// TwinCAT 3 PLC project Tester_QA
// ProgramVersion: 3.1.4024.0
// libraries:
//   AircomLibrary, * (AirCom)
//   VisuElemBase, * (System)
//   Tc2_Standard, * (Beckhoff Automation GmbH)
//   Tc2_SUPS, * (Beckhoff Automation GmbH)
//   Tc2_System, * (Beckhoff Automation GmbH)
//   Tc2_Utilities, * (Beckhoff Automation GmbH)
//   Tc3_Module, * (Beckhoff Automation GmbH)
//   VisuDialogs, * (System)
//   Visu User Mgmt Interfaces,newest,System
//   VisuSymbols,3.5.10.0,System
// project tree:
//   / GlobalTextList.TcGTLO, PlcTask.TcTTO, Visualization Manager.TcVMO (not stored), VISU_TASK.TcTTO
//   GVLs/ GVL_IO.TcGVL, GVL_TesterParams.TcGVL
//   POUs/ MAIN.TcPOU
//   QATester/MainBlock/Chamber/FB/ fbChamber.TcPOU, fbSaveFiles.TcPOU
//   QATester/MainBlock/Chamber/ST/ nCompresorTypes.TcDUT (not stored), nTestType.TcDUT (not stored), stControl.TcDUT, stInOuts.TcDUT, stParamsChamber.TcDUT, stTestParams.TcDUT (not stored)
//   QATester/MainBlock/ fbMainBlock.TcPOU
//   QATester/VISUs/Common/ MeasureCalibration.TcVIS, vSmallChamber.TcVIS, vSmallChamber_WEB.TcVIS, vSmallChamber_v2.TcVIS, vSmallChamber_v2_WEB.TcVIS, vTestPicker.TcVIS
//   QATester/VISUs/Screens/Connected/ vFileSave.TcVIS (not stored), vPlotScreen.TcVIS, vRecipe.TcVIS, vService.TcVIS (not stored)
//   QATester/VISUs/Screens/HMI/ vMainScreen.TcVIS, vStatusScreen.TcVIS, vStatusScreen_v2.TcVIS
//   QATester/VISUs/Screens/WEB/ vMainScreen_WEB.TcVIS, vStatusScreen_v2_WEB.TcVIS, vStatusScreen_WEB.TcVIS
//   QATester/VISUs/TextLists/ txlCompresorTypes.TcTLO, txlTestTypes.TcTLO
//   QATester/VISUs/ vMain.TcVIS, vMain_WEB.TcVIS
// real-time tasks:
//   TASK PlcTask: cycle T#10ms, priority 20, ADS port 350
//   TASK VISU_TASK: cycle T#200000us, priority 30, ADS port 351
//   TASK Task 5: cycle T#10ms, priority 1, ADS port 352
// I/O:
//   DEVICE Device 1 (EtherCAT) (disabled), AmsNetId 5.33.161.102.2.1
//     RIO1 (EK1100) [EK1100 EtherCAT Coupler (2A E-Bus)]
//       DI1 (EL1008) [EL1008 8Ch. Dig. Input 24V, 3ms]
//       DO1 (EL2008) [EL2008 8Ch. Dig. Output 24V, 0.5A]
//       DO2 (EL2008) [EL2008 8Ch. Dig. Output 24V, 0.5A]
//       DO3 (EL2008) [EL2008 8Ch. Dig. Output 24V, 0.5A]
//       AI1 (EL3314) [EL3314 4Ch. Ana. Input Thermocouple (TC)]
//       AI2 (EL3164) [EL3164 4Ch. Ana. Input 0-10V]
//       AI3 (EL3164) [EL3164 4Ch. Ana. Input 0-10V]
//       AI4 (EL3164) [EL3164 4Ch. Ana. Input 0-10V]
// variable links:
//   Tester_QA/Tester_QA Instance <-> Device 1 (EtherCAT)/RIO1 (EK1100)/AI1 (EL3314)
//     PlcTask Inputs/GVL_IO.arstInOuts[{0..3}].iTemperature <-> TC Inputs Channel {1..4}/Value  (4 links)
//   Tester_QA/Tester_QA Instance <-> Device 1 (EtherCAT)/RIO1 (EK1100)/AI2 (EL3164)
//     PlcTask Inputs/GVL_IO.arstInOuts[0].iCurrentRaw <-> AI Standard Channel 1/Value
//     PlcTask Inputs/GVL_IO.arstInOuts[1].iCurrentRaw <-> AI Standard Channel 3/Value
//     PlcTask Inputs/GVL_IO.arstInOuts[2].iCurrentRaw <-> AI Standard Channel 2/Value
//     PlcTask Inputs/GVL_IO.arstInOuts[3].iCurrentRaw <-> AI Standard Channel 4/Value
//   Tester_QA/Tester_QA Instance <-> Device 1 (EtherCAT)/RIO1 (EK1100)/AI3 (EL3164)
//     PlcTask Inputs/GVL_IO.arstInOuts[0].iVoltageRaw <-> AI Standard Channel 1/Value
//     PlcTask Inputs/GVL_IO.arstInOuts[1].iVoltageRaw <-> AI Standard Channel 3/Value
//     PlcTask Inputs/GVL_IO.arstInOuts[2].iVoltageRaw <-> AI Standard Channel 2/Value
//     PlcTask Inputs/GVL_IO.arstInOuts[3].iVoltageRaw <-> AI Standard Channel 4/Value
//   Tester_QA/Tester_QA Instance <-> Device 1 (EtherCAT)/RIO1 (EK1100)/AI4 (EL3164)
//     PlcTask Inputs/GVL_IO.arstInOuts[0].iPressureRaw <-> AI Standard Channel 1/Value
//     PlcTask Inputs/GVL_IO.arstInOuts[1].iPressureRaw <-> AI Standard Channel 3/Value
//     PlcTask Inputs/GVL_IO.arstInOuts[2].iPressureRaw <-> AI Standard Channel 2/Value
//     PlcTask Inputs/GVL_IO.arstInOuts[3].iPressureRaw <-> AI Standard Channel 4/Value
//   Tester_QA/Tester_QA Instance <-> Device 1 (EtherCAT)/RIO1 (EK1100)/DI1 (EL1008)
//     PlcTask Inputs/GVL_IO.arstInOuts[{0..3}].bOverCurrent <-> Channel {1..7 step 2}/Input  (4 links)
//     PlcTask Inputs/GVL_IO.arstInOuts[{0..3}].bSafety <-> Channel 2/Input  (4 links)
//   Tester_QA/Tester_QA Instance <-> Device 1 (EtherCAT)/RIO1 (EK1100)/DO1 (EL2008)
//     PlcTask Outputs/GVL_IO.arstInOuts[{0..3}].bFanON <-> Channel {2..8 step 2}/Output  (4 links)
//     PlcTask Outputs/GVL_IO.arstInOuts[{0..3}].bPowerON <-> Channel {1..7 step 2}/Output  (4 links)
//   Tester_QA/Tester_QA Instance <-> Device 1 (EtherCAT)/RIO1 (EK1100)/DO2 (EL2008)
//     PlcTask Outputs/GVL_IO.arstInOuts[{0..3}].bBottle40l <-> Channel {2..8 step 2}/Output  (4 links)
//     PlcTask Outputs/GVL_IO.arstInOuts[{0..3}].bPressureIn <-> Channel {1..7 step 2}/Output  (4 links)
//   Tester_QA/Tester_QA Instance <-> Device 1 (EtherCAT)/RIO1 (EK1100)/DO3 (EL2008)
//     PlcTask Outputs/GVL_IO.arstInOuts[{0..3}].bEjectPresure <-> Channel {1..7 step 2}/Output  (4 links)
//     PlcTask Outputs/MAIN.fb.bRealease40lTank <-> Channel 2/Output

CONFIGURATION Tester_QA
    RESOURCE PLC ON TwinCAT3
        TASK PlcTask(INTERVAL := T#10ms, PRIORITY := 20);
        TASK VISU_TASK(INTERVAL := T#200000us, PRIORITY := 30);
        PROGRAM MAIN WITH PlcTask : MAIN;
        PROGRAM VisuElems_Visu_Prg WITH VISU_TASK : VisuElems.Visu_Prg;
    END_RESOURCE
END_CONFIGURATION

// ---- QATester/MainBlock/Chamber/ST/stControl.TcDUT
TYPE stControl :
STRUCT
	bStartPerform			 	: BOOL; 		//Wykonanie startu 
	bStartAllow					: BOOL;			//Pozwolenie na start
	bStopPerform				: BOOL;			//Wykonanie stopu
	iSetTest					: nTestType :=nTestType.testEOL;	//Wybrany program
	bChamberBusy				: BOOL;			//Czy komora pracuje
	bTank40Used					: BOOL;			//Czy zbiornik 40l jest używany
	tActualTime					: TIME;			//Czas wymuszenia testu
	bResetChamber				: BOOL;			//Wykonanie resetu po błędzie;
	bChamberResoult				: BOOL;			//Wynik z jakiegokolwiek testu
	sTestResult					: STRING;		//Wynik testu wyświetlany do HMI
END_STRUCT
END_TYPE

// ---- QATester/MainBlock/Chamber/ST/stInOuts.TcDUT
TYPE stInOuts :
STRUCT
	bOverCurrent		AT %I*	: BOOL;			//Przekroczony prąd
	bSafety				AT %I*	: BOOL;			//Obsługa safety
	bPowerON			AT %Q*	: BOOL;			//Załączenie zasilania
	bFanON				AT %Q*	: BOOL;			//Załączenie wentylatora
	bPressureIn			AT %Q*	: BOOL;			//Dobicie ciśnienia do ustalonwej na manometrze wartości
	bBottle40l			AT %Q*	: BOOL;			//Załączenie testu z butlą 40l
	bEjectPresure		AT %Q*	: BOOL;			//Zrzucenie ciśnienia z butli 1l
	bEjectPresure40		AT %Q*	: BOOL;			//Zrzucenie ciśnmienia z butli 40l
	
	iPressureRaw		AT %I* 	: INT;			//Surowa wartość ciśnienia
	iVoltageRaw			AT %I*	: INT;			//Surowa wartość napięcia
	iCurrentRaw			AT %I*	: INT;			//Surowa wartość prądu
	
	rPressure			 		: REAL;			//Wartość ciśnienia
	rVoltage					: REAL;			//Wartość napięcia
	rCurrent					: REAL;			//Wartość prądu
	rTemperature				: REAL;			//Wartość temperatury
	iTemperature		AT %I*	: INT;			//Wartość temperatury
END_STRUCT
END_TYPE

// ---- QATester/MainBlock/Chamber/ST/stParamsChamber.TcDUT
TYPE stParamsChamber :
STRUCT
//Nazwy testów / kompresorów
	sTestName 			: STRING := 'Test';			//Nazwa dla aktuanie wykonywanego testu
	sCompressorName 	: STRING;					//Nazwa dla kompresora
	sErrorDescription	: STRING;					//Opis aktualnego błędu
	sChamberName		: STRING;					//Nazwa komory dla zapisu plików
	sFileDirectory		: STRING;					//Lokalizacja dla zapisu plików
	sFileName			: STRING;					//Nazwa pliku
//Konfigruacja komory
	iCompresorType		: nCompresorTypes := 1;			//Typ kompresora
	iTestNumber			: INT;						//Numer testu
	rMinimalPressure	: REAL;						//Ciśnienie minimalne dla startu komory 
	//stChamberTestParams	:s stTestParams;				//Parametry testu dla komory
	//Parametryzacja zapisu plików
	bSaveToFile			: BOOL;						//Czy zezwolić na zapis do pliku
	iSaveEveryRecords	: INT;						//Wykonaj zapis co ile rekodrów
	iSampleTime0_150	: INT;						//Okres próbkowania do zapisu
	iSampleTime0_1		: INT;						//Okres próbkowania do zapisu
	iSampleTime1_x		: INT;						//Okres próbkowania do zapisu
	sFileCopyLocation	: STRING;					//Gdzie kopoiwać pliki

//Struktury do sterowania skalowaniem wartości fizycznych
	stPressureSens 		: stMeasurementScalingData;	// Parametry skalowania prądu
	stVoltageSens 		: stMeasurementScalingData;	// Parametry skalowania napięcia
	stCurrenteSens 		: stMeasurementScalingData;	// Parametry skalowania prądu
END_STRUCT
END_TYPE

// ---- GVLs/GVL_IO.TcGVL
{attribute 'qualified_only'}
VAR_GLOBAL
	arstInOuts			: ARRAY[0..3] OF stInOuts;
END_VAR

// ---- GVLs/GVL_TesterParams.TcGVL
{attribute 'qualified_only'}
VAR_GLOBAL PERSISTENT
	arTestParams		: ARRAY[0..3] OF stTestParams;
	arstParams			: ARRAY[0..3] OF stParamschamber;
END_VAR
VAR_GLOBAL
	arstControl			: ARRAY[0..3] OF stControl;
	stData				: stAircomTimeStruct;
END_VAR

// ---- POUs/MAIN.TcPOU
PROGRAM MAIN
VAR
	fb : fbMainBlock;
	fbAircomTime : fbDateAndTimeCalc;
	saveDataPresistent : WritePersistentData;
	fbSavePerform	: TON;
	i : INT;
	arTestParams		: ARRAY[0..3] OF stTestParams;
	arstParams			: ARRAY[0..3] OF stParamschamber;
	bSaveData	: BOOL;
	bInit	: BOOL;
END_VAR

IF NOT bInit THEN
	MEMCPY(destAddr:= ADR(arTestParams), srcAddr:=ADR(GVL_TesterParams.arTestParams)  ,n:= SIZEOF(stTestParams)*4);
	MEMCPY(destAddr:= ADR(arstParams), srcAddr:=ADR(GVL_TesterParams.arstParams)  ,n:= SIZEOF(stParamschamber)*4);
	bInit := TRUE;
END_IF
fb(arstControl	:=GVL_TesterParams.arstControl,
	arstParams	:= GVL_TesterParams.arstParams,
	arstInOuts	:= GVL_IO.arstInOuts,
	stChamberTestParams := GVL_TesterParams.arTestParams);
fbAircomTime();

bSaveData	S= (MEMCMP(pBuf1 := ADR(GVL_TesterParams.arTestParams),pBuf2:= ADR(arTestParams), n:= SIZEOF(stTestParams)*4) <> 0) OR (MEMCMP(pBuf1 := ADR(GVL_TesterParams.arstParams),pBuf2:= ADR(arstParams), n:= SIZEOF(stParamschamber)*4) <> 0);
	
fbSavePerform(IN:=bSaveData ,PT:=T#300S);		
IF fbSavePerform.Q THEN
	saveDataPresistent(NETID:='',PORT:=851,START:=TRUE,TMOUT:=T#2S);
	bSaveData R= TRUE;
	MEMCPY(destAddr:= ADR(arTestParams), srcAddr:=ADR(GVL_TesterParams.arTestParams)  ,n:= SIZEOF(stTestParams)*4);
	MEMCPY(destAddr:= ADR(arstParams), srcAddr:=ADR(GVL_TesterParams.arstParams)  ,n:= SIZEOF(stParamschamber)*4);
ELSE
	saveDataPresistent(START:=FALSE);
END_IF

END_PROGRAM

// ---- QATester/MainBlock/fbMainBlock.TcPOU
FUNCTION_BLOCK fbMainBlock
VAR_INPUT
END_VAR
VAR_OUTPUT
END_VAR
VAR_IN_OUT
	arstControl			: ARRAY[0..3] OF stControl;
	arstParams			: ARRAY[0..3] OF stParamschamber;
	arstInOuts			: ARRAY[0..3] OF stInOuts;
	stChamberTestParams : ARRAY[0..3] OF stTestParams;
END_VAR
VAR
	arFbChamber		: ARRAY[0..3] OF fbChamber;
	i			: INT;
	bTankBusy		: BOOL;
	bRealease40lTank	AT %Q* : BOOL;
END_VAR

//Bloki funkcyjne

FOR i := 0 TO 3 DO
	arstControl[i].bStartAllow := NOT arstControl[i].bChamberBusy;		
	arFbChamber[i](stControl:=arstControl[i],stInOuts:=arstInOuts[i],stParams:=arstParams[i],stChamberTestParams:=stChamberTestParams[arstParams[i].iCompresorType],stTime:=GVL_Aircom.stAC_DT_Data);
END_FOR

END_FUNCTION_BLOCK

// ---- QATester/MainBlock/Chamber/FB/fbChamber.TcPOU
FUNCTION_BLOCK fbChamber
VAR_INPUT
END_VAR
VAR_OUTPUT
END_VAR
VAR_IN_OUT
	stControl				: stControl;
	stInOuts 				: stInOuts;
	stParams				: stParamsChamber;
	stChamberTestParams		: stTestParams;
	stTime					: stAircomTimeStruct;	//Struktura czasu
END_VAR
VAR
	//Bloki skalujące
	fbPressureScaller 		:fbAnalogMeasurement;	//Blok skalujący ciśnienie
	fbVoltageScaller	 	:fbAnalogMeasurement;	//Blok skalujący napięcie
	fbCurrentScaller 		:fbAnalogMeasurement;	//Blok skalujący prąd
	iWorkStep : INT;
	//Detekcja prądu
	fbCurrentCheckDelayer	: TON;					//Zwłoka dla wykrywania prądu minimalnego
	//Test EOL
	fbTestTimerEOL			: TON;					//Licznik czasu trwania testu EOL
	bEolTestResult			: BOOL;					//Wynik z testu EOL
	//Test Performance
	fbTestTimerPerformance	: TON;					//Licznik czasu trwania testu Wydajnoiściowego
	bPerfornamceTestResult	: BOOL;					//Wynik z testu Wydajnościowego
	//Test Hour
	fbTestTimerHour	: TON;							//Licznik czasu trwania testu Wydajnoiściowego
	bHourTestResult	: BOOL;							//Wynik z testu Wydajnościowego
	bPressureObtainedHour :BOOL;					//Pierwsza faza zakończona osiągnięto ciśnienie testowe
	//Test Whole
	iWorkStepWhole	: INT;							//Kroki programowe dla testu całościowego
	fbTestTimerWholeI	: TON;							//Licznik czasu I test całkowity
	fbTestTimerWholeII	: TON;							//Licznik czasu II test całkowity
	//Test Under Presure
	bUnderPresureTestResult : BOOL;					//Wynik testu pod ciśnieniem
	rStartUnderPresureLastPresureRecord : REAL;		//Save value of presure before test
	fbUnderPresureTestTimer	: TON;							//Licznik czasu dla tesu pod ciśnieniem
	//Test Cyclic 30
	iCyclicLoopVariable 		: INT;				//Wariable for calculate of cyclic loops
	fbTestTimerCyclic30			: TON;				//Licznik czasu trwania testu cyklicznego 30
	bCyclic30TestResult			: BOOL;				//Wynik testu cyklicznego x30
	fbTestTimerCyclic30On		: TON;				//Timer dla obsługi testu
	bFirstCycle30				: BOOL;				//First cycle indefiner
	iWorkStepTest30				: INT;				//Workstep dla testu cyklicznego 70
	//Test Cyclic 70
	fbTestTimerCyclic70			: TON;				//Licznik czasu trwania testu cyklicznego 30
	bCyclic70TestResult			: BOOL;				//Wynik testu cyklicznego x30
	fbTestTimerCyclic70On		: TON;				//Timer dla obsługi testu
	bFirstCycle70				: BOOL;				//First cycle indefiner
	iWorkStepTest70				: INT;				//Workstep dla testu cyklicznego 70
	//Zmienne do obsługi zapisu plików
	sData						: STRING;			//Data dopisana do lokalizacji
	sDate						: STRING;			//Data rozpoczęcia testu
	sTime						: STRING;			//Godzina rozpoczęcia testu
	sTestName					: STRING;			//Nazwa Test
	sFirstLine					: STRING;			//Dane do zapisu w pierwszej linijce
	sDataString					: STRING(5000);			//dane z pomiarami
	sDataStringTmp				: STRING(5000);			//dane z pomiarami
	sDataStringTmpSave			: STRING(5000);			//Dane do zapisu
	sActualTestTime				: STRING;			//Aktualny czas testu
	sActualPresure				: STRING;			//Aktualna wartość ciśnienia
	sActualVoltage				: STRING;			//Aktualna wartość napięcia
	sActualCurrent				: STRING;			//Aktualna wartość prądu
	sActualTemperature			: STRING;			//Aktualna wartość temperatury
	fbTestTime					: TON;				//Czas wykonywania testu
	iSaveFileRecords			: INT;				//Aktualnie zapisane rekody do zapisu pliku
	iSaveFileRecordsTmp			: INT;				//Zapisana ilość rekordów w tablicy do zapisu (zmienne skopiowane)
	bCreateFile					: BOOL;				//Wymueszenie utworzenia nowego pliku
	bInsertNewStartRows			: BOOL;				//Wymuszenie wstawienia pierwszych 2 wierszy 
	bSavePerform				: BOOL;				//Wykonaj zapis do pliku
	bCopyArray					: BOOL;				//Przygotowanie buforów do zapisu
	arTmpData					: ARRAY[0..1000] OF STRING;	//Tablica z zmiennymi
	arTmpDataCpy				: ARRAY[0..1000] OF STRING;	//Tablica z zmiennymi skopiowanymi
	fbFileOpen					: FB_FileOpen;		//Funkcja dla otwierania pliku
	fbFileClose					: FB_FileClose;		//Funkcja dla zamknięcia pliku
	fbFileWrite					: FB_FileWrite;		//Funkcja dla zapisu pliku
	sFileNameToSave				: STRING;			//Nazwa do zapisu pliku
	bReadyToWrite				: BOOL;				//Zezwolenie na zapis do pliku
	bReadyToClose				: BOOL;				//Zezwolenie na zamknięcie pliku
	bFileSaveError				: BOOL;				//Błąd podczas tworzenie zapisów
	iSampleRecorder				: INT;				//Obsługa samplingu
	fbTestTimer					: TON;				//Obsługa czasu trwania testu
	sTimeRep					: STRING;			//Zmienna dla obsługi czasu godzina 
	fbRiseEdgeError				: R_TRIG;
	iSaveCalc					: INT;				// zmienna pomocnicza podczas zapisu danych
	bRecordTaker				: BOOL;				//Zmienna dla obsługi zbierania danych
	wRecordCalc					: DWORD;			//Zmienna dla lcizenia czasu testu
	bFileCopy					: BOOL;				//Zmienna wykorzystywana podczas kopiowania plików
	fbFileSave					: fbSaveFiles;		//Save files save
	fbFileSaveCopy				: fbSaveFiles;		//Save files save
	//Zmienne dla obsługi rysowania grafów
	arPlotPresure				: ARRAY[0..1000] OF REAL;
	arPlotVoltage				: ARRAY[0..1000] OF REAL;
	arPlotCurrent				: ARRAY[0..1000] OF REAL;
	iPlotRecordCounter			: INT;
	sStepDescription			: STRING;
	iPlotFilter					: INT;
	sFileCopyCommand			: STRING(1000);
	sTemString					: STRING;
	bTEST: BOOL;
	sDirCopy: STRING;
	sPathCopy:STRING;
	iLastWorkStep: INT;
	fbRestON: TON;
END_VAR

ACT_Background();
CASE iWorkStep OF
 0: 				//Inicalizacja
 	iWorkStep := 5;
	stParams.sErrorDescription :='';
	fbTestTimer(IN:=FALSE);
	stInOuts.bFanON := stInOuts.bPowerON := stInOuts.bEjectPresure40 := stInOuts.bEjectPresure := stInOuts.bBottle40l := stInOuts.bPressureIn := FALSE;
 5:					//Idle
 	sStepDescription := 'Chamber Idle';
	stParams.sTestName:= '';
	stControl.tActualTime := T#40D;
	bUnderPresureTestResult R= bCyclic70TestResult R= bCyclic30TestResult R= bPerfornamceTestResult R= bEolTestResult R= stControl.bStartPerform;
 	IF stControl.bStartPerform AND stControl.iSetTest >= 20 AND stInOuts.rPressure <= stParams.rMinimalPressure THEN
		iWorkStep := 6;
		stControl.sTestResult := '';
		stControl.tActualTime := stTime.tActualTime;
	ELSIF stControl.bStartPerform AND stControl.iSetTest = nTestType.testEOL AND stInOuts.rPressure <= stParams.rMinimalPressure THEN
		iWorkStep := stControl.iSetTest;
		stControl.bStartPerform := FALSE;
		bInsertNewStartRows := TRUE;
	ELSIF stControl.bStartPerform THEN
		stInOuts.bEjectPresure := TRUE;
		sStepDescription := 'Presure droping';
	END_IF
 6:
 	sStepDescription := 'Wait for bottle 40l';
 	IF stControl.iSetTest = nTestType.testEOL OR NOT stControl.bStartPerform THEN
		iWorkStep := 5;
		stControl.bStartPerform := FALSE;
		stControl.tActualTime := T#40D;
	END_IF
 	IF stControl.bStartAllow THEN
		bInsertNewStartRows := TRUE;
		bUnderPresureTestResult := bCyclic70TestResult := bCyclic30TestResult := bPerfornamceTestResult := bEolTestResult := FALSE;
		iWorkStep := stControl.iSetTest;
		bFirstCycle70 := bFirstCycle30 := TRUE;
		stControl.bStartAllow := FALSE;
		stControl.bStartPerform := FALSE;
	END_IF

 10: 				//EOL Test
 	stParams.sTestName:= 'EOL_Test';
	ACT_EolTest();
	IF bEolTestResult THEN
		iWorkStep := 1000;
		bEolTestResult:= FALSE;
	END_IF
 20:				//Performance Test
	stParams.sTestName:= 'Performance_Test';
 	ACT_PerformanceTest();
	IF bPerfornamceTestResult THEN
		iWorkStep := 1000;
		bPerfornamceTestResult := FALSE;
	END_IF
 30:				//Hour Test
 	stParams.sTestName:= 'Hour_Test';
 	ACT_HourTest();
	IF bHourTestResult THEN
		iWorkStep := 1000;
		bHourTestResult := FALSE;
	END_IF
 40:				//Whole Test
 	stParams.sTestName:= 'Full_Test';
 	Act_WholeTest();
 50:				//Cyclic x30 Test
 	stParams.sTestName:= 'Cyclic_x30_Test';
 	ACT_Cyclic30Test();
	IF bCyclic30TestResult THEN
		iWorkStep := 1000;
		bCyclic30TestResult := FALSE;
	END_IF
 60:				//Cyclic x70 Test
 	stParams.sTestName:= 'Cyclic_x70_Test';
 	ACT_Cyclic70Test();
	IF bCyclic70TestResult THEN
		iWorkStep := 1000;
		bCyclic70TestResult := FALSE;
	END_IF
 200:				// Błąd
 	//Wysterowanie Timerów i zmiennch
 	fbTestTimerEOL(IN:=FALSE);fbTestTimerPerformance(IN:=FALSE);fbTestTimerHour(IN:=FALSE);fbTestTimerWholeI(IN:=FALSE);
	fbTestTimerWholeII(IN:=FALSE);fbUnderPresureTestTimer(IN:=FALSE);fbTestTimerCyclic30(IN:=FALSE);fbTestTimerCyclic30On(IN:=FALSE);
	fbTestTimerCyclic70(IN:=FALSE);fbTestTimerCyclic70On(IN:=FALSE);
	bUnderPresureTestResult := bCyclic70TestResult := bCyclic30TestResult := bPerfornamceTestResult := bEolTestResult := stInOuts.bFanON := stInOuts.bPowerON := stInOuts.bEjectPresure := stInOuts.bBottle40l := stInOuts.bPressureIn := FALSE;
 	stControl.tActualTime := T#40D;
	stControl.sTestResult := 'Faliure';
 	fbTestTimer(IN:=FALSE);
	stControl.bStartAllow := stControl.bStartPerform := FALSE;
	IF stInOuts.rPressure >= stParams.rMinimalPressure THEN
		stInOuts.bEjectPresure40 := TRUE;
		sStepDescription := 'Error pressure droping';
	ELSE
		stControl.bTank40Used := FALSE;
		stInOuts.bEjectPresure40 := FALSE;
		sStepDescription := 'Wait for reset';
	END_IF
 	IF stControl.bResetChamber THEN
		iWorkStep:=0;
		stControl.bResetChamber := FALSE;
		bFileCopy := TRUE;
	END_IF
 1000:				//Przygotowanie komory do następnego testu
 	stInOuts.bEjectPresure40 S= (bPerfornamceTestResult OR bHourTestResult OR bCyclic70TestResult OR bCyclic30TestResult);
	stInOuts.bEjectPresure S= bEolTestResult;
	iWorkStepTest70 := iWorkStepTest30 := iWorkStepWhole := 0;
	sStepDescription := 'Presure droping';
	stControl.sTestResult := 'DONE';
 	IF stInOuts.rPressure <= stParams.rMinimalPressure THEN
		stControl.tActualTime := T#40D;
		stInOuts.bEjectPresure40 := stInOuts.bEjectPresure := FALSE;
		bUnderPresureTestResult := bCyclic70TestResult := bPerfornamceTestResult := bHourTestResult := bCyclic30TestResult := FALSE;
		iWorkStep := 0;
		bFileCopy := TRUE;
	END_IF
END_CASE

ACTION ACT_Background:
//Obsługa zatrzymania
IF stControl.bChamberBusy AND stControl.bStopPerform THEN
	iWorkStep := 200;
	stControl.bStopPerform := FALSE;
	stParams.sErrorDescription:='Test detained';
END_IF
fbRestON(IN:=stControl.bResetChamber,Pt:=T#200MS);
IF fbRestON.Q THEN
	stControl.bResetChamber  := FALSE;
END_IF
//Skalowanie pomiarów Ciśnienia/Napięcia/Prądu
	fbPressureScaller(rIn:=stInOuts.iPressureRaw,stMeasureScalingData:=stParams.stPressureSens,tStalaCzasowa:=T#10MS,rOutFiltered=>stInOuts.rPressure);
	fbVoltageScaller(rIn:=stInOuts.iVoltageRaw,stMeasureScalingData:=stParams.stVoltageSens,tStalaCzasowa:=T#10MS,rOutFiltered=>stInOuts.rVoltage);
	fbCurrentScaller (rIn:=stInOuts.iCurrentRaw,stMeasureScalingData:=stParams.stCurrenteSens,tStalaCzasowa:=T#10MS,rOutFiltered=>stInOuts.rCurrent);
	stInOuts.rTemperature := stInOuts.iTemperature/10;
//Obsługa Safety
IF stInOuts.bSafety	THEN
	stParams.sErrorDescription := 'Emergency button pressed';
	iWorkStep := 200;
END_IF
//Obsługa daty
sData := CONCAT(WORD_TO_STRING(stTime.stTimeStruct.wYear),'_');
sData := CONCAT(sData,WORD_TO_STRING(stTime.stTimeStruct.wMonth));
//Obsługa zbiornika
	stControl.bTank40Used := iWorkStep >= 20; 		//Określenie czy zbiornik 40l jest wykorzystywany
//Obsługa sekwencji
	stControl.bChamberBusy := (iWorkStep >=10);		//Określenie czy komora wykonuje prace
	stControl.bStartPerform R= (iWorkStep > 6);	//Kasowanie wymuszenia staru po rozpoczęciu nowej pracy
//Sprawowanie kontroli nad prądem minimalnym
	fbCurrentCheckDelayer(IN:=stInOuts.bPowerON,PT:=REAL_TO_TIME(stChamberTestParams.rMinimalCurrentCheckDelay*1000));
	IF fbCurrentCheckDelayer.Q AND (stChamberTestParams.rMinimalCurrentLimit > stInOuts.rCurrent) THEN
		stParams.sErrorDescription := 'Minimal current obtain error';
		iWorkStep := 200;
	END_IF
//Zapis Pliku 
sDate := CONCAT(CONCAT(CONCAT(CONCAT(WORD_TO_STRING(stTime.stTimeStruct.wYear),'_'),WORD_TO_STRING(stTime.stTimeStruct.wMonth)),'_'),WORD_TO_STRING(stTime.stTimeStruct.wDay));
sTimeRep := CONCAT(CONCAT(CONCAT(CONCAT(WORD_TO_STRING(stTime.stTimeStruct.wHour),'_'),WORD_TO_STRING(stTime.stTimeStruct.wMinute)),'_'),WORD_TO_STRING(stTime.stTimeStruct.wSecond));	
sDate := CONCAT(CONCAT(sDate,'_'),sTimeRep);
IF stControl.bChamberBusy AND stParams.bSaveToFile THEN
	ACT_DataSampling();
ELSE
	wRecordCalc := 0;
END_IF
IF stControl.bChamberBusy AND (stParams.sErrorDescription = '') THEN
	ACT_GraphWriter();
	sStepDescription := 'Work in progress';
ELSIF iPlotRecordCounter <> 0 THEN
	iPlotRecordCounter := 0;
	MEMSET(destAddr:=ADR(arPlotPresure),fillByte:=16#00,n:=SIZEOF(arPlotPresure[0])*1000);
	MEMSET(destAddr:=ADR(arPlotVoltage),fillByte:=16#00,n:=SIZEOF(arPlotVoltage[0])*1000);
	MEMSET(destAddr:=ADR(arPlotCurrent),fillByte:=16#00,n:=SIZEOF(arPlotCurrent[0])*1000);
ELSIF NOT stControl.bChamberBusy AND stParams.sErrorDescription = '' THEN
	sStepDescription := 'Idle';
ELSIF stParams.sErrorDescription <> '' THEN
	sStepDescription := 'Chamber Error';
END_IF
//Timer dla obsługi aktualnego czasu
fbTestTime(IN:=stControl.bChamberBusy,PT:=T#5D);
//Wyniki z testów
stControl.bChamberResoult := bUnderPresureTestResult OR bCyclic70TestResult OR bCyclic30TestResult OR bPerfornamceTestResult OR bEolTestResult;
END_ACTION

ACTION ACT_Cyclic30Test:
//Nowa sekwencja
//Obliczanie czasu trwania testu
fbTestTimer(IN:=stINOuts.bPowerON,PT:=T#10D);
//Sekwencja
CASE iWorkStepTest30 OF
	0:	//Test wydajnościowy
		bCyclic30TestResult:= FALSE;
		iCyclicLoopVariable := 0;
		ACT_PerformanceTest();
		IF bPerfornamceTestResult THEN
			iWorkStepTest30 := 10;
		END_IF
	10: //Krok statowy spuszczenie ciśnienia
		bPerfornamceTestResult := FALSE;
		stInOuts.bEjectPresure40 := stInOuts.bEjectPresure := TRUE;
		IF stInOuts.rPressure <= stPArams.rMinimalPressure THEN
			iWorkStepTest30 := 20;
		END_IF
	20:	//Oczekiwanie na dostarczenie do układu ciśnienia po zakończeniu czasu oczekiwania
		stInOuts.bEjectPresure40 := stInOuts.bEjectPresure := FALSE;
		fbTestTimerCyclic30On(IN:=TRUE,PT:=REAL_TO_TIME(stChamberTestParams.rTestCycle30CoolingTime*1000));
		IF fbTestTimerCyclic30On.Q OR bFirstCycle70 THEN
			stInOuts.bPressureIn := TRUE;
		END_IF
		IF stInOuts.bPressureIn AND ABS((stInOuts.rPressure - stChamberTestParams.rStartPresureCycle30Test) < 0.1) THEN
			stInOuts.bPressureIn := FALSE;
			iWorkStepTest70 := 30;
		END_IF
	30:	//Sprawdzenie ciśnienia
		IF stInOuts.bPressureIn AND ((stInOuts.rPressure - stChamberTestParams.rStartPresureCycle30Test) > 0.2) AND stChamberTestParams.bCheckStartPresureCycle70 THEN
			iWorkStep:= 200;
			stInOuts.bFanON := stInOuts.bPowerON := FALSE;
			stInOuts.bEjectPresure40 := stInOuts.bEjectPresure := TRUE;
			stParams.sErrorDescription := 'Wrong start pressure';
			fbTestTimerPerformance(IN:=FALSE);
		ELSE
			iWorkStepTest30 := 40;
		END_IF
	40:	// Rozpoczęcie pierwszej sekwencji
		stInOuts.bFanON := stInOuts.bPowerON := TRUE;
		fbTestTimerCyclic30On(IN:= stInOuts.bPowerON,PT:=REAL_TO_TIME(stChamberTestParams.rTestCycle30LimitTime)*1000);
		IF fbTestTimerCyclic30On.Q AND stChamberTestParams.rPresureToObtainCycle30Test <= stInOuts.rPressure THEN
			iCyclicLoopVariable := iCyclicLoopVariable + 1;
			bFirstCycle30 := FALSE;
			stInOuts.bEjectPresure40 := stInOuts.bEjectPresure := TRUE;
			stInOuts.bPowerON := FALSE;
			fbTestTimerCyclic30On(IN:=FALSE);
			fbTestTimerCyclic30(IN:=FALSE);
			stInOuts.bPowerON := FALSE;
			IF iCyclicLoopVariable >=30 THEN
				iWorkStepTest30 := 50;
				//
				iCyclicLoopVariable := 0;
				bFirstCycle30:= TRUE;
			ELSE
				iWorkStepTest30 := 10;
			END_IF
		END_IF
		IF (fbTestTimerPerformance.Q AND stChamberTestParams.rPresureToObtainCycle70Test >= stInOuts.rPressure) THEN
			iWorkStep:= 200;
			stInOuts.bFanON := stInOuts.bPowerON := FALSE;
			stInOuts.bEjectPresure40 := stInOuts.bEjectPresure := TRUE;
			stParams.sErrorDescription := 'Compressor did not obtain set pressure in limited time';
			bPerfornamceTestResult := FALSE;
			fbTestTimerPerformance(IN:=FALSE);
		END_IF
	50://Zakończenie testu i wykonanie nowego testu wydajnościowego
		bCyclic30TestResult:= FALSE;
		iCyclicLoopVariable := 0;
		ACT_PerformanceTest();
		IF bPerfornamceTestResult THEN
			iWorkStepTest30 := 60;
		END_IF
	60: //Wydanie danych o zakończonej poprawnej pracy
		bCyclic30TestResult := TRUE;
		bPerfornamceTestResult := FALSE;
		fbTestTimerPerformance(IN:=FALSE);
END_CASE
END_ACTION

ACTION ACT_Cyclic70Test:
//Nowa sekwencja
//Obliczanie czasu trwania testu
fbTestTimer(IN:=stINOuts.bPowerON,PT:=T#10D);
//Sekwencja
CASE iWorkStepTest70 OF
	0:	//Test wydajnościowy
		bCyclic70TestResult:= FALSE;
		iCyclicLoopVariable := 0;
		ACT_PerformanceTest();
		IF bPerfornamceTestResult THEN
			iWorkStepTest70 := 10;
		END_IF
	10: //Krok statowy spuszczenie ciśnienia
		bPerfornamceTestResult := FALSE;
		stInOuts.bEjectPresure40 := stInOuts.bEjectPresure := TRUE;
		IF stInOuts.rPressure <= stPArams.rMinimalPressure THEN
			iWorkStepTest70 := 20;
		END_IF
	20:	//Oczekiwanie na dostarczenie do układu ciśnienia po zakończeniu czasu oczekiwania
		stInOuts.bEjectPresure40 := stInOuts.bEjectPresure := FALSE;
		fbTestTimerCyclic70On(IN:=TRUE,PT:=REAL_TO_TIME(stChamberTestParams.rTestCycle70CoolingTime*1000));
		IF fbTestTimerCyclic70On.Q OR bFirstCycle70 THEN
			stInOuts.bPressureIn := TRUE;
		END_IF
		IF stInOuts.bPressureIn AND ABS((stInOuts.rPressure - stChamberTestParams.rStartPresureCycle70Test) < 0.1) THEN
			stInOuts.bPressureIn := FALSE;
			iWorkStepTest70 := 30;
		END_IF
	30:	//Sprawdzenie ciśnienia
		IF stInOuts.bPressureIn AND ((stInOuts.rPressure - stChamberTestParams.rStartPresureCycle70Test) > 0.2) AND stChamberTestParams.bCheckStartPresureCycle70 THEN
			iWorkStep:= 200;
			stInOuts.bFanON := stInOuts.bPowerON := FALSE;
			stInOuts.bEjectPresure40 := stInOuts.bEjectPresure := TRUE;
			stParams.sErrorDescription := 'Wrong start pressure';
			fbTestTimerPerformance(IN:=FALSE);
		ELSE
			iWorkStepTest70 := 40;
		END_IF
	40:	// Rozpoczęcie pierwszej sekwencji
		stInOuts.bFanON := stInOuts.bPowerON := TRUE;
		fbTestTimerCyclic70On(IN:= stInOuts.bPowerON,PT:=REAL_TO_TIME(stChamberTestParams.rTestCycle70LimitTime)*1000);
		IF fbTestTimerCyclic70On.Q AND stChamberTestParams.rPresureToObtainCycle70Test <= stInOuts.rPressure THEN
			iCyclicLoopVariable := iCyclicLoopVariable + 1;
			bFirstCycle70 := FALSE;
			stInOuts.bEjectPresure40 := stInOuts.bEjectPresure := TRUE;
			stInOuts.bPowerON := FALSE;
			fbTestTimerCyclic70On(IN:=FALSE);
			fbTestTimerCyclic70(IN:=FALSE);
			stInOuts.bPowerON := FALSE;
			IF iCyclicLoopVariable >=70 THEN
				iWorkStepTest70 := 50;
				//
				iCyclicLoopVariable := 0;
				bFirstCycle70:= TRUE;
			ELSE
				iWorkStepTest70 := 10;
			END_IF
		END_IF
		IF (fbTestTimerPerformance.Q AND stChamberTestParams.rPresureToObtainCycle70Test >= stInOuts.rPressure) THEN
			iWorkStep:= 200;
			stInOuts.bFanON := stInOuts.bPowerON := FALSE;
			stInOuts.bEjectPresure40 := stInOuts.bEjectPresure := TRUE;
			stParams.sErrorDescription := 'Compressor did not obtain set pressure in limited time';
			bPerfornamceTestResult := FALSE;
			fbTestTimerPerformance(IN:=FALSE);
		END_IF
	50://Zakończenie testu i wykonanie nowego testu wydajnościowego
		bCyclic70TestResult:= FALSE;
		iCyclicLoopVariable := 0;
		ACT_PerformanceTest();
		IF bPerfornamceTestResult THEN
			iWorkStepTest70 := 60;
		END_IF
	60: //Wydanie danych o zakończonej poprawnej pracy
		bCyclic70TestResult := TRUE;
		bPerfornamceTestResult := FALSE;
		fbTestTimerPerformance(IN:=FALSE);
END_CASE
END_ACTION

ACTION ACT_DataSampling:
//Resetowanie licznika czasu testu podczas zmiany testu np w teście penym aby na nowo wyzwolić nowe próbkowania
IF iWorkStep <> iLastWorkStep THEN
	iLastWorkStep := iWorkStep;
	wRecordCalc := 0;
END_IF
//Liczenie kolejnych wywołań progrmau
wRecordCalc := wRecordCalc +1;
//Przygotowywanie zmiennych nagłówkowych
IF bInsertNewStartRows AND stParams.sTestName <> '' THEN
	//Przygotowanie ścieżki pliku z nazwą
	sFileNameToSave:= '';
	sFileNameToSave:= CONCAT(sFileNameToSave,sDate);
	sFileNameToSave:= CONCAT(sFileNameToSave,'_');
	sFileNameToSave:= CONCAT(sFileNameToSave,stParams.sChamberName);
	sFileNameToSave:= CONCAT(sFileNameToSave,'_');
	sFileNameToSave:= CONCAT(sFileNameToSave,sTestName);
	sFileNameToSave:= CONCAT(sFileNameToSave,'_');
	sFileNameToSave:= CONCAT(sFileNameToSave,stParams.sTestName);
	sFileNameToSave:= CONCAT(sFileNameToSave,'.csv');
	bInsertNewStartRows := FALSE;
	//Tworzenie nagłówków 
	sDataStringTmp := CONCAT(sDate,',');
	sDataStringTmp := CONCAT(sDataStringTmp,stParams.sChamberName);
	sDataStringTmp := CONCAT(sDataStringTmp,',');
	sDataStringTmp := CONCAT(sDataStringTmp,stParams.sFileName);
	sDataStringTmp := CONCAT(sDataStringTmp,',');
	sDataStringTmp := CONCAT(sDataStringTmp,sTestName);
	sDataStringTmp := CONCAT(sDataStringTmp,'$R');
	sDataStringTmp := CONCAT(sDataStringTmp,'Czas [s],Prąd [A],Ciśnienie [bar],Napięcie [V],Temperatura [°C]$R');
	sDataString := sDataStringTmp;
	iSaveFileRecords := 2;
END_IF
//Cykliczne przygotowyawanie zmiennych
IF stParams.sErrorDescription = '' THEN
	iSampleRecorder := iSampleRecorder + 1;
	bRecordTaker := (*iSampleRecorder >= 1;*)(iSampleRecorder >= stParams.iSampleTime0_150/10 AND  wRecordCalc  <=  15) OR (iSampleRecorder >= stParams.iSampleTime0_1/10 AND  wRecordCalc  > 15 AND  wRecordCalc  <=  100) 
		OR (iSampleRecorder >= stParams.iSampleTime1_x/10 AND  wRecordCalc  >  100);
	IF bRecordTaker THEN
		sActualTestTime 	:= REAL_TO_STRING(TIME_TO_REAL(fbTestTime.ET)/1000);
		sActualPresure 		:= REAL_TO_STRING(stInOuts.rPressure);					//Przepisanie wartości ciśnienia
		sActualVoltage 		:= REAL_TO_STRING(stInOuts.rVoltage);					//Przepisanie wartości napięcia
		sActualCurrent 		:= REAL_TO_STRING(stInOuts.rCurrent);					//Przepisanie wartości prądu
		sActualTemperature 	:= REAL_TO_STRING(stInOuts.rTemperature);											//Przepisanie wartości temperatury
		//Przygotowanie zmiennych cyklicznych do zapisu oraz przemieszczenie danych do bufora
		sDataStringTmp 		:= CONCAT(sActualTestTime,',');					//Zapisanie aktualnego czasu 
		sDataStringTmp 		:= CONCAT(sDataStringTmp,sActualCurrent);			//Dopisanie wartości prądu
		sDataStringTmp 		:= CONCAT(sDataStringTmp,',');						//Przypisanie odstępu format CSV
		sDataStringTmp 		:= CONCAT(sDataStringTmp,sActualPresure);			//Dopisanie wartości ciśnienia
		sDataStringTmp 		:= CONCAT(sDataStringTmp,',');						//Przypisanie odstępu format CSV
		sDataStringTmp 		:= CONCAT(sDataStringTmp,sActualVoltage);			//Dopisanie wartości napięcia
		sDataStringTmp 		:= CONCAT(sDataStringTmp,',');						//Przypisanie odstępu format CSV
		sDataStringTmp 		:= CONCAT(sDataStringTmp,sActualTemperature);		//Dopisanie wartości temperatury
		sDataStringTmp 		:= CONCAT(sDataStringTmp,'$R');						//Dopisanie znaku enter
		CONCAT2(pSrcString1:=ADR(sDataString),pSrcString2:=ADR(sDataStringTmp),pDstString:=ADR(sDataString),nDstSize:=SIZEOF(sDataString));
		iSaveFileRecords 	:= iSaveFileRecords + 1;
		iSampleRecorder 	:= 0;
	END_IF
END_IF
//Wykonanie zapisu oraz uporzątkowanie zmiennych/buforów
fbRiseEdgeError(CLK:=(stParams.sErrorDescription <> '' OR iWorkStep = 1000));
fbFileSave.bExecute S= ((iSaveFileRecords >= stParams.iSaveEveryRecords) OR fbRiseEdgeError.Q ) AND NOT fbFileSave.bBusy;
fbFileSaveCopy.bExecute S= ((iSaveFileRecords >= stParams.iSaveEveryRecords) OR fbRiseEdgeError.Q ) AND NOT fbFileSave.bBusy;
IF fbFileSave.bDone AND fbFileSave.bDone THEN
	iSaveFileRecords := 0;
	fbFileSave.bExecute R= TRUE;
	fbFileSaveCopy.bExecute R= TRUE;
	sDataString := '';
END_IF
//Wykonanie funkcji zapisu
fbFileSave(
	sFileNameToSave:=sFileNameToSave,
	sDataStringTmpSave:=sDataString,
	sFileDirectory:=CONCAT(stParams.sFileDirectory,sData));
fbFileSaveCopy(
	sFileNameToSave:=sFileNameToSave,
	sDataStringTmpSave:=sDataString,
	sFileDirectory:=CONCAT(stParams.sFileCopyLocation,sData));
END_ACTION

ACTION ACT_EolTest:
fbTestTimer(IN:=stINOuts.bPowerON,PT:=T#10D);
stInOuts.bEjectPresure40 := stInOuts.bEjectPresure := stInOuts.bBottle40l := stInOuts.bPressureIn := FALSE;
stInOuts.bFanON := stInOuts.bPowerON := TRUE;
fbTestTimerEOL(IN:= stInOuts.bPowerON,PT:=REAL_TO_TIME(stChamberTestParams.rTestEolLimitTime*1000));
IF fbTestTimerEOL.Q THEN
	iWorkStep:= 200;
	stInOuts.bFanON := stInOuts.bPowerON := FALSE;
	stInOuts.bEjectPresure := TRUE;
	stParams.sErrorDescription := 'Compressor did not obtain set pressure in limited time';
	bEolTestResult := FALSE;
	fbTestTimerEOL(IN:=FALSE);
END_IF
IF stChamberTestParams.rPresureToObtainEOLTest < stInOuts.rPressure THEN
	bEolTestResult := TRUE;
	fbTestTimerEOL(IN:=FALSE);
END_IF
END_ACTION

ACTION ACT_GraphWriter:
//ZApis informacji odnośnie grafów na wizualizacji
iPlotFilter := iPlotFilter + 1;
IF iPlotFilter >= 5 THEN
	arPlotPresure[iPlotRecordCounter] := stInOuts.rPressure;
	arPlotVoltage[iPlotRecordCounter] := stInOuts.rVoltage;
	arPlotCurrent[iPlotRecordCounter] := stInOuts.rCurrent;
	iPlotRecordCounter := iPlotRecordCounter + 1;
	iPlotFilter := 0;
	IF iPlotRecordCounter >= 500 THEN
		iPlotRecordCounter := 0;
		MEMSET(destAddr:=ADR(arPlotPresure),fillByte:=16#00,n:=SIZEOF(arPlotPresure[0])*1000);
		MEMSET(destAddr:=ADR(arPlotVoltage),fillByte:=16#00,n:=SIZEOF(arPlotVoltage[0])*1000);
		MEMSET(destAddr:=ADR(arPlotCurrent),fillByte:=16#00,n:=SIZEOF(arPlotCurrent[0])*1000);
	END_IF
END_IF
END_ACTION

ACTION ACT_HourTest:
fbTestTimer(IN:=stINOuts.bPowerON,PT:=T#10D);
stInOuts.bEjectPresure40 := stInOuts.bEjectPresure := stInOuts.bPressureIn := FALSE;
stInOuts.bBottle40l := stInOuts.bFanON := stInOuts.bPowerON := TRUE;
fbTestTimerHour(IN:= (stChamberTestParams.rPressureToObtainHourTest<=stInOuts.rPressure),PT:=REAL_TO_TIME(stChamberTestParams.rTestHourTime*1000));
bPressureObtainedHour S= (stChamberTestParams.rPressureToObtainHourTest<=stInOuts.rPressure);
IF bPressureObtainedHour AND ABS(stInOuts.rPressure-stChamberTestParams.rPressureToObtainHourTest) > stChamberTestParams.rTestHourPressureMaximalTolerance THEN
	iWorkStep:= 200;
	stInOuts.bFanON := stInOuts.bPowerON := FALSE;
	stInOuts.bEjectPresure40 := stInOuts.bEjectPresure := TRUE;
	stParams.sErrorDescription := 'Pressure deviation too high';
	bHourTestResult := FALSE;
	fbTestTimerHour(IN:= FALSE);
END_IF
IF fbTestTimerPerformance.Q THEN
	bHourTestResult := TRUE;
	bPressureObtainedHour R= TRUE;
	fbTestTimerHour(IN:= FALSE);
END_IF
END_ACTION

ACTION ACT_PerformanceTest:
fbTestTimerPerformance(IN:= stInOuts.bPowerON,PT:=REAL_TO_TIME(stChamberTestParams.rTest300SecTime*1000));
fbTestTimer(IN:=stINOuts.bPowerON,PT:=T#10D);
stInOuts.bEjectPresure40 := stInOuts.bEjectPresure := stInOuts.bPressureIn := FALSE;
stInOuts.bBottle40l := stInOuts.bFanON := stInOuts.bPowerON := TRUE;
IF (fbTestTimerPerformance.Q AND stChamberTestParams.rPresureToObtainPerformanceTest >= stInOuts.rPressure) THEN
	iWorkStep:= 200;
	stInOuts.bFanON := stInOuts.bPowerON := FALSE;
	stInOuts.bEjectPresure40 := stInOuts.bEjectPresure := TRUE;
	stParams.sErrorDescription := 'Compressor did not obtain set pressure in limited time';
	bPerfornamceTestResult := FALSE;
	fbTestTimerPerformance(IN:=FALSE);
ELSIF (stChamberTestParams.rCurrentLimitPerformacneTest < stInOuts.rCurrent) THEN
	iWorkStep:= 200;
	stInOuts.bFanON := stInOuts.bPowerON := FALSE;
	stInOuts.bEjectPresure40 := stInOuts.bEjectPresure := TRUE;
	stParams.sErrorDescription := 'Current to high';
	bPerfornamceTestResult := FALSE;
	fbTestTimerPerformance(IN:=FALSE);
END_IF
IF fbTestTimerPerformance.Q AND stChamberTestParams.rPresureToObtainPerformanceTest <= stInOuts.rPressure THEN
	bPerfornamceTestResult := TRUE;
	stInOuts.bPowerON := stInOuts.bFanON := FALSE;
	fbTestTimerPerformance(IN:=FALSE);
END_IF
END_ACTION

ACTION ACT_TestUnderPressure:
fbTestTimer(IN:=stINOuts.bPowerON,PT:=T#10D);
IF stInOuts.rPressure < (stChamberTestParams.rTestUnderPresureSetPresure - stChamberTestParams.rTestUnderPresureCloseTolerance) THEN
	stInOuts.bEjectPresure40 := stInOuts.bEjectPresure := FALSE;
	stInOuts.bPressureIn := stInOuts.bBottle40l := TRUE;
ELSE
	stInOuts.bPressureIn := FALSE;
END_IF
IF ABS(stInOuts.rPressure - stChamberTestParams.rTestUnderPresureSetPresure) < stChamberTestParams.rTestUnderPresureStartTolerance AND NOT stInOuts.bPressureIn THEN
	stInOuts.bPowerON := TRUE;
	rStartUnderPresureLastPresureRecord := stInOuts.rPressure;
END_IF

IF stInOuts.bPowerON THEN
	fbUnderPresureTestTimer(IN:=TRUE,PT:=REAL_TO_TIME(stChamberTestParams.rTestUnderPresureTime*1000));
	IF (stInOuts.rPressure - stChamberTestParams.rTestUnderPresureSetPresure) > stChamberTestParams.rTestUnderPresureMinimalIncrease THEN
		bUnderPresureTestResult := TRUE;
	ELSIF fbUnderPresureTestTimer.Q THEN
		iWorkStep:= 200;
		stInOuts.bFanON := stInOuts.bPowerON := FALSE;
		stInOuts.bEjectPresure40 := stInOuts.bEjectPresure := TRUE;
		stParams.sErrorDescription := 'Start under presure failt to obtain presure increase in definied time';
		bUnderPresureTestResult := FALSE;
		fbUnderPresureTestTimer(IN:=FALSE);
	END_IF
END_IF
END_ACTION

ACTION ACT_WholeTest:
CASE iWorkStepWhole OF 
	0:	//Test wydajnościowy
		ACT_PerformanceTest();
		IF bPerfornamceTestResult THEN
			iWorkStepWhole := 5;
			bPerfornamceTestResult := FALSE;
		END_IF
	5:
		stInOuts.bEjectPresure := stInOuts.bEjectPresure40 := TRUE;
		IF stInOuts.rPressure <= stParams.rMinimalPressure THEN
			stInOuts.bEjectPresure40 := stInOuts.bEjectPresure := FALSE;
			iWorkStepWhole := 10;
		END_IF
	10:	//Oczekiwanie 
		fbTestTimerWholeI(IN:=TRUE,PT:=REAL_TO_TIME(stChamberTestParams.rTestCoolingTimeFullStepI*1000));
		IF fbTestTimerWholeI.Q THEN
			iWorkStepWhole := 20;
			fbTestTimerWholeI(IN:=FALSE);
		END_IF
	20:	//Test godzinny
		ACT_HourTest();
		IF bHourTestResult THEN
			iWorkStepWhole := 25;
			bHourTestResult := FALSE;
		END_IF
	25: //Test pod ciśnieniem
		ACT_TestUnderPressure();
		IF bUnderPresureTestResult THEN
			iWorkStepWhole := 30;
			bUnderPresureTestResult := FALSE;
		END_IF
	30:
		stInOuts.bEjectPresure := stInOuts.bEjectPresure40 := TRUE;
		IF stInOuts.rPressure <= stParams.rMinimalPressure THEN
			stInOuts.bEjectPresure40 := stInOuts.bEjectPresure := FALSE;
			iWorkStepWhole := 35;
		END_IF
	35:	//Oczekiwanie II
		fbTestTimerWholeII(IN:=TRUE,PT:=REAL_TO_TIME(stChamberTestParams.rTestCoolingTimeFullStepII*1000));
		IF fbTestTimerWholeII.Q THEN
			iWorkStepWhole := 40;
			fbTestTimerWholeII(IN:=FALSE);
		END_IF
	40:
		ACT_PerformanceTest();
		IF bPerfornamceTestResult THEN
			iWorkStep:=1000;
			bPerfornamceTestResult := FALSE;
			iWorkStepWhole := 0;
		END_IF
	



END_CASE
END_ACTION

END_FUNCTION_BLOCK

// ---- QATester/MainBlock/Chamber/FB/fbSaveFiles.TcPOU
FUNCTION_BLOCK fbSaveFiles
VAR_INPUT
	bExecute					: BOOL;				//Wywołanie funkcji
	sData						: STRING;			//DATA
	sFileNameToSave				: STRING;			//Nazwa do zapisu pliku
	sDataStringTmpSave			: STRING(5000);		//Dane do zapisu
	sFileDirectory				: STRING;			//Scieżka do zapisu pliku
END_VAR
VAR_OUTPUT
	bBusy						: BOOL;				//Funkcja podczas pracy
	bDone						: BOOL;				//Opercja została wykonana
	bError						: BOOL;				//Błąd podaczas zapisu
END_VAR
VAR_IN_OUT

END_VAR
VAR
	fbFileOpen					: FB_FileOpen;		//Funkcja dla otwierania pliku
	fbFileClose					: FB_FileClose;		//Funkcja dla zamknięcia pliku
	fbFileWrite					: FB_FileWrite;		//Funkcja dla zapisu pliku
	fbCreateDir					: FB_CreateDir;		//Tworzenie Folder
	iWorkStep					: INT;				//Int dla obsługi kolejkowania 
	fbTriggerExecute			: R_TRIG;			//Reakcja na polecenie wykonania funkcji
	sFilePath					: STRING;
END_VAR

fbTriggerExecute(CLK:=bExecute);
sFilePath := CONCAT(sFileDirectory,'\');
sFilePath := CONCAT(sFilePath,sFileNameToSave);
CASE iWorkStep OF
	0://Krok inicializujący
		fbFileClose(bExecute:=FALSE);
		fbFileWrite(bExecute:=FALSE);
		fbFileOpen(bExecute:=FALSE);
		fbCreateDir(bExecute:=FALSE);
		IF fbTriggerExecute.Q THEN
			iWorkStep:= 5;
			bBusy:=TRUE;
			bDone := FALSE;
		END_IF
	5: //Tworzenie folderu
		fbCreateDir(sNetId:='',
			sPathName:=sFileDirectory,
			ePath:=PATH_GENERIC,
			bExecute:=TRUE,
			tTimeout:=T#2S);
	IF NOT fbCreateDir.bBusy  THEN
		IF fbCreateDir.nErrId = 16#723 OR fbCreateDir.nErrId = 1804 THEN		//Sprawdzenie czy folder istnieje
			iWorkStep:= 10;
		ELSE
			fbCreateDir(bExecute:=FALSE);
		END_IF
		
	END_IF
	10:
		fbFileOpen(sNetId:='',
			sPathName:=sFilePath,
			nMode:=FOPEN_MODEAPPEND,
			ePath:=PATH_GENERIC,
			bExecute:=TRUE,
			tTimeout:=T#2S);
		IF  NOT fbFileOpen.bBusy THEN
			iWorkStep:= 20;
		END_IF	
	20:
		fbFileWrite(sNetId:='',
			hFile:=fbFileOpen.hFile,
			pWriteBuff:=ADR(sDataStringTmpSave),
			cbWriteLen:=SIZEOF(BYTE)*LEN2(pString:=ADR(sDataStringTmpSave)),
			bExecute:=TRUE,
			tTimeout:=T#2S);
		IF  NOT fbFileWrite.bBusy THEN
			iWorkStep:= 30;
		END_IF		
	30:
		fbFileClose(sNetId:='',
			hFile:=fbFileOpen.hFile,
			bExecute:=TRUE,
			tTimeout:=T#2S);
		IF  NOT fbFileClose.bBusy THEN
			iWorkStep:= 40;
		END_IF
	40:
		bDone := TRUE;
		iWorkStep:= 50;
	50:
	 	IF NOT bexecute THEN
			iWorkStep:= 0;
			bDone := FALSE;
			bBusy := FALSE;
		END_IF
END_CASE

END_FUNCTION_BLOCK

// ---- GlobalTextList.TcGTLO
TEXTLIST GlobalTextList
  842 = '%.0f'
  209 = '%.1f'
  240 = '%.2f'
  978 = '%b'
  905 = '%b.0'
  856 = '%d'
  100 = '%f'
  991 = '%f.1'
  798 = '%s'
  302 = '1 Hour test'
  205 = '300 sec'
  393 = '< Act'
  1794 = 'Actual'
  996 = 'Actual '
  499 = 'Actual chamber'
  409 = 'Actual Chamber'
  952 = 'Admin'
  360 = 'Amper'
  155 = 'Analog settings'
  490 = 'Bar'
  479 = 'Bottle release \nconformation pressure'
  189 = 'Bottle release \nconformation pressure [Bar]'
  28 = 'Bottle release conformation pressure'
  516 = 'Cancel change'
  9 = 'Chamber'
  361 = 'Chamber\nStatus'
  663 = 'Chamber 1'
  656 = 'Chamber 2'
  910 = 'Chamber 3'
  78 = 'Chamber 4'
  734 = 'Check start presure'
  200 = 'Checkbox'
  150 = 'Complete Test'
  68 = 'Compresor Type'
  591 = 'Compresor type'
  166 = 'Compressor Type'
  105 = 'Connect valve'
  633 = 'Cooling time [s]'
  71 = 'Current'
  828 = 'Current limit'
  505 = 'Current limit [A]'
  373 = 'Cycle time [s]'
  521 = 'Cycli x30 Test'
  438 = 'Cycli x70 Test'
  137 = 'Eject presure'
  498 = 'Eject presure 1l'
  43 = 'Eject presure 40l'
  493 = 'Eng'
  729 = 'EOL Test'
  984 = 'Error'
  454 = 'fbChamber.stControl.bChamberResoult'
  535 = 'File Name'
  906 = 'File name'
  543 = 'File operations'
  655 = 'File operations error'
  879 = 'File remote path'
  568 = 'File Save \nScreen'
  694 = 'File settings'
  554 = 'First cooling time'
  613 = 'First cooling time [s]'
  214 = 'Home \nScreen'
  590 = 'Home Screen'
  1759 = 'I point'
  2580 = 'II point'
  419 = 'Logout'
  654 = 'Manual Operations'
  446 = 'Maximal Presure decrease [bar]'
  826 = 'Maximal start time [s]'
  474 = 'Maxmial diffrence in presure [bar]'
  2651 = 'Measured'
  17 = 'Minimal current check time [s]'
  369 = 'Minimal current [A]'
  456 = 'Minimal presure increase [bar]'
  547 = 'New'
  61 = 'None'
  690 = 'Operation Desc'
  517 = 'Operator'
  395 = 'Path'
  702 = 'Performance'
  926 = 'Performance Test'
  863 = 'Plot \nScreen'
  585 = 'Presure'
  691 = 'Presure Input'
  943 = 'Presure to obtain'
  104 = 'Presure to obtain [bar]'
  67 = 'Presure valve turn off [bar]'
  898 = 'QA'
  2034 = 'Raw'
  184 = 'Recipe'
  466 = 'Recipe \nScreen'
  608 = 'Reset Perform'
  367 = 'Sampling time'
  101 = 'Sampling time 0 - 1 [s]'
  1173 = 'Sampling time 0 - 150 [ms] | [ms]'
  1002 = 'Sampling time 0 - 300 [s]'
  866 = 'Sampling time 1 - 300 [s]'
  887 = 'Sampling time 150 - 1000 [ms] | [ms]'
  975 = 'Sampling time t  > 1 [s]'
  152 = 'Sampling time x  > 1 [s] | [ms]'
  758 = 'Save every'
  791 = 'Save every n records'
  620 = 'Save perform'
  576 = 'Saving Error'
  92 = 'Second cooling time'
  624 = 'Second cooling time [s]'
  796 = 'Service'
  907 = 'Service \nScreen'
  861 = 'Set pressure to start [bar]'
  727 = 'Set pressure to start [s]'
  577 = 'Set presure to start [bar]'
  867 = 'Start Perform'
  315 = 'Start under presure'
  603 = 'Stop Perform'
  380 = 'Temperature'
  765 = 'Test name'
  786 = 'Test result'
  857 = 'Test time'
  942 = 'Test time [s]'
  956 = 'Test Type'
  294 = 'Themp'
  536 = 'Turn off presure valve before [bar]'
  701 = 'Turn On Power'
  179 = 'User'
  972 = 'User\nLogin'
  2421 = 'Value'
  106 = 'Volt'
  578 = 'Voltage'
  1883 = '^^ Set NEW ^^'
  1045 = '^^^ Confirm change !!! ^^^'
END_TEXTLIST

// ---- QATester/VISUs/Common/MeasureCalibration.TcVIS
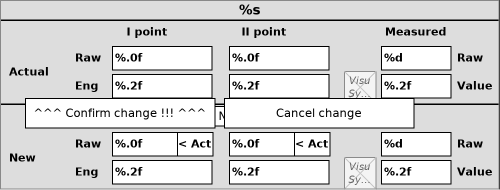
VISUALIZATION MeasureCalibration  // 500x190
VAR_IN_OUT
	stMeasureData:stMeasurementScalingData;
END_VAR
VAR_INPUT
	diAnalogIn:DINT;
	MeasureName:STRING;
END_VAR
VAR
	rRaw1:REAL;
	rRaw2:REAL:= 32767;
	rEng1:REAL;
	rEng2:REAL;
	bConfirmation:BOOL:=FALSE;
END_VAR
    Rectangle (0,20 500x84)
    Rectangle (112,46 100x24), "%.0f", text variable: stMeasureData.rScalingRawValue_I, input disabled if: TRUE
    Label (72,46 40x24), "Raw"
    Rectangle (112,74 100x24), "%.2f", text variable: stMeasureData.rScalingEngValue_I, input disabled if: TRUE
    Label (72,74 40x24), "Eng"
    Label (112,20 70x24), "I point"
    Rectangle (229,46 100x24), "%.0f", text variable: stMeasureData.rScalingRawValue_II, input disabled if: TRUE
    Rectangle (229,74 100x24), "%.2f", text variable: stMeasureData.rScalingEngValue_II, input disabled if: TRUE
    Label (229,20 70x24), "II point"
    Image (344,71 32x32), image: VisuSymbols.Symbols.ArrowBoldRight
    Label (381,20 70x24), "Measured"
    Rectangle (381,74 70x24), "%.2f", text variable: ( (DINT_TO_REAL(diAnalogIn) - stMeasureData.rScalingRawValue_I)/ ( LIMIT(0.1,(stMeasureData.rScalingRawValue_II - stMeasureData.rScalingRawValue_I),999999999999)))*( stMeasureData.rScalingEngValue_II - stMeasureData.rScalingEngValue_I)+stMeasureData.rScalingEngValue_I, input disabled if: TRUE
    Rectangle (381,46 70x24), "%d", text variable: diAnalogIn, input disabled if: TRUE
    Label (454,46 40x24), "Raw"
    Label (454,74 40x24), "Value"
    Rectangle (0,104 500x85)
    Rectangle (112,132 68x24), "%.0f", text variable: rRaw1
        OnMouseClick: write rRaw1 via Default, title 'New Raw I value', format %.0f
    Label (72,132 40x24), "Raw"
    Rectangle (112,160 100x24), "%.2f", text variable: rEng1
        OnMouseClick: write rEng1 via Default, title 'New Eng I value', format %.2f
    Label (72,160 40x24), "Eng"
    Rectangle (229,132 68x24), "%.0f", text variable: rRaw2
        OnMouseClick: write rRaw2 via Default, title 'New Raw II value', format %.0f
    Rectangle (229,160 100x24), "%.2f", text variable: rEng2
        OnMouseClick: write rEng2 via Default, title 'New Eng II value', format %.2f
    Image (344,157 32x32), image: VisuSymbols.Symbols.ArrowBoldRight
    Rectangle (381,160 70x24), "%.2f", text variable: ( (DINT_TO_REAL(diAnalogIn) - rRaw1)/ (LIMIT(1,(rRaw2 - rRaw1),9999999999999) ) ) * ( rEng2 - rEng1)+ rEng1, input disabled if: TRUE
    Rectangle (381,132 70x24), "%d", text variable: diAnalogIn, input disabled if: TRUE
    Label (454,132 40x24), "Raw"
    Label (454,160 40x24), "Value"
    Label (6,146 40x24), "New"
    Label (6,60 40x24), "Actual"
    RoundedRectangle (113,106 216x20), "^^ Set NEW ^^", invisible if: bConfirmation
        toggle bConfirmation
    RoundedRectangle (177,132 36x24), "< Act"
        OnMouseClick: execute { rRaw1:= DINT_TO_REAL(diAnalogIn); }
    RoundedRectangle (294,132 36x24), "< Act"
        OnMouseClick: execute { rRaw2 := DINT_TO_REAL(diAnalogIn); }
    RoundedRectangle (25,98 190x30), "^^^ Confirm change !!! ^^^", invisible if: NOT bConfirmation
        OnMouseClick: execute {
            stMeasureData.rScalingEngValue_I := rEng1;
            stMeasureData.rScalingEngValue_II := rEng2;
            stMeasureData.rScalingRawValue_I := rRaw1;
            stMeasureData.rScalingRawValue_II := rRaw2;
            bConfirmation:= FALSE;
        }
    RoundedRectangle (224,98 190x30), "Cancel change", invisible if: NOT bConfirmation
        OnMouseClick: execute { bConfirmation:= FALSE; }
    Rectangle (0,0 500x20), "%s", text variable: MeasureName
END_VISUALIZATION

// ---- QATester/VISUs/Common/vSmallChamber.TcVIS
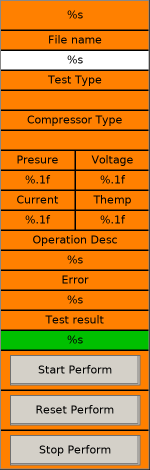
VISUALIZATION vSmallChamber  // 150x470
VAR_IN_OUT
	stParams : stParamsChamber;
	fbChamber : fbChamber;
	stControl : stControl;
END_VAR
    Rectangle (0,390 150x40)
    Rectangle (0,350 150x40)
    Rectangle (0,50 150x20), "%s", text variable: fbChamber.sTestName
        OnMouseClick: write the text variable via VisuDialogs.Keypad
    Rectangle (0,30 150x20), "File name"
    Button (10,355 130x30), "Start Perform", pressed state: stControl.bStartPerform, input disabled if: stControl.bChamberBusy
        OnMouseClick: toggle stControl.bStartPerform
    Rectangle (0,90 150x20), text list: 'txlTestTypes', text index: fbChamber.stControl.iSetTest
    Rectangle (0,70 150x20), "Test Type"
    Rectangle (0,110 150x20), "Compressor Type"
    Rectangle (0,130 150x20), text list: 'txlCompresorTypes', text index: fbChamber.stParams.iCompresorType
    Rectangle (0,150 75x20), "Presure"
    Rectangle (75,150 75x20), "Voltage"
    Rectangle (0,170 75x20), "%.1f", text variable: fbChamber.stInOuts.rPressure
    Rectangle (75,170 75x20), "%.1f", text variable: fbChamber.stInOuts.rVoltage
    Rectangle (0,190 75x20), "Current"
    Rectangle (0,210 75x20), "%.1f", text variable: fbChamber.stInOuts.rVoltage
    Rectangle (0,230 150x20), "Operation Desc"
    Rectangle (0,250 150x20), "%s", text variable: fbChamber.sStepDescription
    Rectangle (0,310 150x20), "Test result"
    Rectangle (0,330 150x20), "%s", text variable: stControl.sTestResult, colour toggle: stControl.sTestResult <> 'DONE'
    Rectangle (0,270 150x20), "Error"
    Rectangle (0,290 150x20), "%s", text variable: stParams.sErrorDescription
    Rectangle (0,0 150x30), "%s", text variable: stParams.sChamberName
    Button (10,395 130x30), "Reset Perform", pressed state: stControl.bResetChamber AND stParams.sErrorDescription = ''
        OnMouseClick: toggle stControl.bResetChamber
    Rectangle (75,190 75x20), "Themp"
    Rectangle (75,210 75x20), "%.1f", text variable: fbChamber.stInOuts.rTemperature
    Rectangle (0,430 150x40)
    Button (10,435 130x30), "Stop Perform", pressed state: stControl.bStopPerform, input disabled if: NOT stControl.bChamberBusy
        OnMouseClick: toggle stControl.bStopPerform
END_VISUALIZATION

// ---- QATester/VISUs/Common/vSmallChamber_WEB.TcVIS
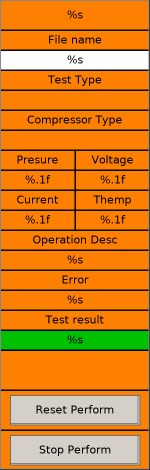
VISUALIZATION vSmallChamber_WEB  // 150x470
VAR_IN_OUT
	stParams : stParamsChamber;
	fbChamber : fbChamber;
	stControl : stControl;
END_VAR
    Rectangle (0,390 150x40)
    Rectangle (0,350 150x40)
    Rectangle (0,50 150x20), "%s", text variable: fbChamber.sTestName
        OnMouseClick: write the text variable via VisuDialogs.Keypad
    Rectangle (0,30 150x20), "File name"
    Rectangle (0,90 150x20), text list: 'txlTestTypes', text index: fbChamber.stControl.iSetTest
    Rectangle (0,70 150x20), "Test Type"
    Rectangle (0,110 150x20), "Compressor Type"
    Rectangle (0,130 150x20), text list: 'txlCompresorTypes', text index: fbChamber.stParams.iCompresorType
    Rectangle (0,150 75x20), "Presure"
    Rectangle (75,150 75x20), "Voltage"
    Rectangle (0,170 75x20), "%.1f", text variable: fbChamber.stInOuts.rPressure
    Rectangle (75,170 75x20), "%.1f", text variable: fbChamber.stInOuts.rVoltage
    Rectangle (0,190 75x20), "Current"
    Rectangle (0,210 75x20), "%.1f", text variable: fbChamber.stInOuts.rVoltage
    Rectangle (0,230 150x20), "Operation Desc"
    Rectangle (0,250 150x20), "%s", text variable: fbChamber.sStepDescription
    Rectangle (0,310 150x20), "Test result"
    Rectangle (0,330 150x20), "%s", text variable: stControl.sTestResult, colour toggle: stControl.sTestResult <> 'DONE'
    Rectangle (0,270 150x20), "Error"
    Rectangle (0,290 150x20), "%s", text variable: stParams.sErrorDescription
    Rectangle (0,0 150x30), "%s", text variable: stParams.sChamberName
    Button (10,395 130x30), "Reset Perform", pressed state: stControl.bResetChamber AND stParams.sErrorDescription = ''
        OnMouseClick: toggle stControl.bResetChamber
    Rectangle (75,190 75x20), "Themp"
    Rectangle (75,210 75x20), "%.1f", text variable: fbChamber.stInOuts.rTemperature
    Rectangle (0,430 150x40)
    Button (10,435 130x30), "Stop Perform", pressed state: stControl.bStopPerform, input disabled if: NOT stControl.bChamberBusy
        OnMouseClick: toggle stControl.bStopPerform
END_VISUALIZATION

// ---- QATester/VISUs/Common/vSmallChamber_v2.TcVIS
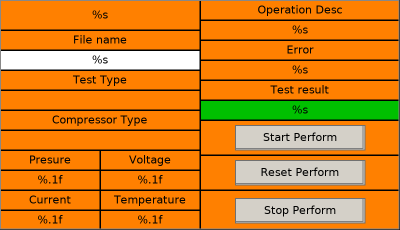
VISUALIZATION vSmallChamber_v2  // 400x230
VAR_IN_OUT
	stParams : stParamsChamber;
	fbChamber : fbChamber;
	stControl : stControl;
END_VAR
    Rectangle (200,155 200x35)
    Rectangle (200,120 200x35)
    Rectangle (0,50 200x20), "%s", text variable: fbChamber.sTestName
        OnMouseClick: write the text variable via VisuDialogs.Keypad
    Rectangle (0,30 200x20), "File name"
    Button (235,125 130x25), "Start Perform"
        OnMouseClick: toggle stControl.bStartPerform
    Rectangle (0,90 200x20), text list: 'txlTestTypes', text index: fbChamber.stControl.iSetTest
    Rectangle (0,70 200x20), "Test Type"
    Rectangle (0,110 200x20), "Compressor Type"
    Rectangle (0,130 200x20), text list: 'txlCompresorTypes', text index: fbChamber.stParams.iCompresorType
    Rectangle (0,150 100x20), "Presure"
    Rectangle (100,150 100x20), "Voltage"
    Rectangle (0,170 100x20), "%.1f", text variable: fbChamber.stInOuts.rPressure
    Rectangle (100,170 100x20), "%.1f", text variable: fbChamber.stInOuts.rVoltage
    Rectangle (0,190 100x20), "Current"
    Rectangle (0,210 100x20), "%.1f", text variable: fbChamber.stInOuts.rVoltage
    Rectangle (200,0 200x20), "Operation Desc"
    Rectangle (200,20 200x20), "%s", text variable: fbChamber.sStepDescription
    Rectangle (200,80 200x20), "Test result"
    Rectangle (200,100 200x20), "%s", text variable: stControl.sTestResult, colour toggle: stControl.sTestResult <> 'DONE'
    Rectangle (200,40 200x20), "Error"
    Rectangle (200,60 200x20), "%s", text variable: stParams.sErrorDescription
    Rectangle (0,0 200x30), "%s", text variable: stParams.sChamberName
    Button (235,160 130x25), "Reset Perform"
        OnMouseClick: toggle stControl.bResetChamber
    Rectangle (100,210 100x20), "%.1f", text variable: fbChamber.stInOuts.rTemperature
    Rectangle (100,190 100x20), "Temperature"
    Rectangle (200,190 200x40)
    Button (235,198 130x25), "Stop Perform"
        OnMouseClick: toggle stControl.bStopPerform
END_VISUALIZATION

// ---- QATester/VISUs/Common/vSmallChamber_v2_WEB.TcVIS
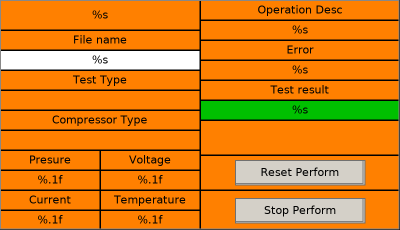
VISUALIZATION vSmallChamber_v2_WEB  // 400x230
VAR_IN_OUT
	stParams : stParamsChamber;
	fbChamber : fbChamber;
	stControl : stControl;
END_VAR
    Rectangle (200,155 200x35)
    Rectangle (200,120 200x35)
    Rectangle (0,50 200x20), "%s", text variable: fbChamber.sTestName
        OnMouseClick: write the text variable via VisuDialogs.Keypad
    Rectangle (0,30 200x20), "File name"
    Rectangle (0,90 200x20), text list: 'txlTestTypes', text index: fbChamber.stControl.iSetTest
    Rectangle (0,70 200x20), "Test Type"
    Rectangle (0,110 200x20), "Compressor Type"
    Rectangle (0,130 200x20), text list: 'txlCompresorTypes', text index: fbChamber.stParams.iCompresorType
    Rectangle (0,150 100x20), "Presure"
    Rectangle (100,150 100x20), "Voltage"
    Rectangle (0,170 100x20), "%.1f", text variable: fbChamber.stInOuts.rPressure
    Rectangle (100,170 100x20), "%.1f", text variable: fbChamber.stInOuts.rVoltage
    Rectangle (0,190 100x20), "Current"
    Rectangle (0,210 100x20), "%.1f", text variable: fbChamber.stInOuts.rVoltage
    Rectangle (200,0 200x20), "Operation Desc"
    Rectangle (200,20 200x20), "%s", text variable: fbChamber.sStepDescription
    Rectangle (200,80 200x20), "Test result"
    Rectangle (200,100 200x20), "%s", text variable: stControl.sTestResult, colour toggle: stControl.sTestResult <> 'DONE'
    Rectangle (200,40 200x20), "Error"
    Rectangle (200,60 200x20), "%s", text variable: stParams.sErrorDescription
    Rectangle (0,0 200x30), "%s", text variable: stParams.sChamberName
    Button (235,160 130x25), "Reset Perform"
        OnMouseClick: toggle stControl.bResetChamber
    Rectangle (100,210 100x20), "%.1f", text variable: fbChamber.stInOuts.rTemperature
    Rectangle (100,190 100x20), "Temperature"
    Rectangle (200,190 200x40)
    Button (235,198 130x25), "Stop Perform"
        OnMouseClick: toggle stControl.bStopPerform
END_VISUALIZATION

// ---- QATester/VISUs/Common/vTestPicker.TcVIS
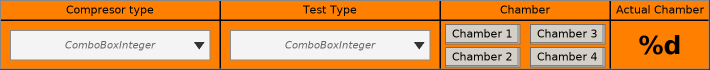
VISUALIZATION vTestPicker  // 710x70
VAR_IN_OUT
	iCompressorPick : nCompresorTypes;
	iTestType		: nTestType;
	iActualChamber	: INT;
	arControl		: ARRAY[0..3] OF stControl;
END_VAR
    Rectangle (0,20 220x50)
    ComboBoxInteger (10,30 200x30), variable: iCompressorPick, input disabled if: arControl[iActualChamber].bChamberBusy OR arControl[iActualChamber].bStartPerform, text list: 'txlCompresorTypes'
    Rectangle (0,0 220x20), "Compresor type"
    Rectangle (220,20 220x50)
    Rectangle (220,0 220x20), "Test Type"
    ComboBoxInteger (230,30 200x30), variable: iTestType, input disabled if: arControl[iActualChamber].bChamberBusy OR arControl[iActualChamber].bStartPerform, text list: 'txlTestTypes'
    Rectangle (440,0 170x20), "Chamber"
    Rectangle (440,20 170x50)
    Rectangle (610,0 100x20), "Actual Chamber"
    Rectangle (610,20 100x50), "%d", text variable: iActualChamber + 1
    Button (445,24 75x20), "Chamber 1"
        OnMouseClick: execute { iActualChamber := 0; }
    Button (530,24 75x20), "Chamber 3"
        OnMouseClick: execute { iActualChamber := 2; }
    Button (445,47 75x20), "Chamber 2"
        OnMouseClick: execute { iActualChamber := 1; }
    Button (530,47 75x20), "Chamber 4"
        OnMouseClick: execute { iActualChamber := 3; }
END_VISUALIZATION

// ---- QATester/VISUs/Screens/Connected/vPlotScreen.TcVIS
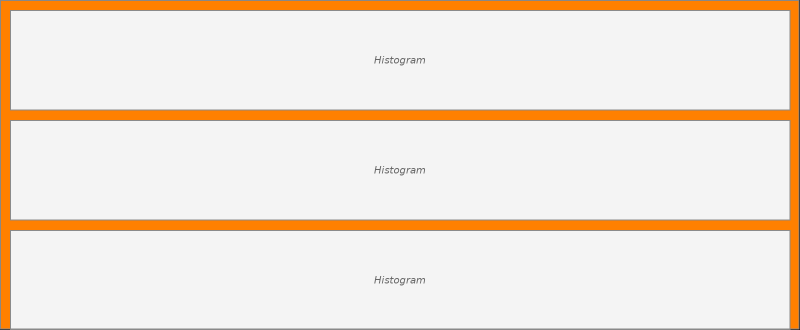
VISUALIZATION vPlotScreen  // 800x330
VAR_IN_OUT
	stControl : stControl;
	fbChamber	: fbChamber;
END_VAR
    Rectangle (0,0 800x330)
    Histogram (10,10 780x100), scale format: %.1f, scale 0..5
        p518627256: Bar
        p1518820177: fbChamber.arPlotPresure
        p102497268: fbChamber.arPlotPresure
        p788070771: ARRAY [0..1000] OF REAL
    Histogram (10,120 780x100), scale format: %.1f, scale 8..14
        p518627256: Volt
        p1518820177: fbChamber.arPlotVoltage
        p102497268: fbChamber.arPlotVoltage
        p788070771: ARRAY [0..1000] OF REAL
    Histogram (10,230 780x100), scale format: %.1f, scale 0..15
        p518627256: Amper
        p1518820177: fbChamber.arPlotCurrent
        p102497268: fbChamber.arPlotCurrent
        p788070771: ARRAY [0..1000] OF REAL
END_VISUALIZATION

// ---- QATester/VISUs/Screens/Connected/vRecipe.TcVIS
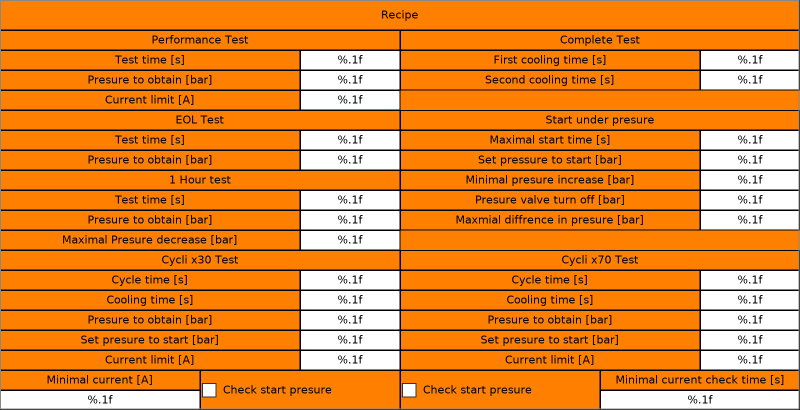
VISUALIZATION vRecipe  // 800x410
VAR_IN_OUT
	fbChamber 	: fbChamber;
	stChamberTestParams	: stTestParams;
END_VAR
    Rectangle (200,370 200x40)
    Rectangle (0,0 800x30), "Recipe"
    Rectangle (0,30 400x20), "Performance Test"
    Rectangle (0,50 300x20), "Test time [s]"
    Rectangle (0,70 300x20), "Presure to obtain [bar]"
    Rectangle (0,90 300x20), "Current limit [A]"
    Rectangle (0,110 400x20), "EOL Test"
    Rectangle (0,130 300x20), "Test time [s]"
    Rectangle (0,150 300x20), "Presure to obtain [bar]"
    Rectangle (0,190 300x20), "Test time [s]"
    Rectangle (0,170 400x20), "1 Hour test"
    Rectangle (0,210 300x20), "Presure to obtain [bar]"
    Rectangle (0,230 300x20), "Maximal Presure decrease [bar]"
    Rectangle (400,50 300x20), "First cooling time [s]"
    Rectangle (400,30 400x20), "Complete Test"
    Rectangle (400,70 300x20), "Second cooling time [s]"
    Rectangle (400,110 400x20), "Start under presure"
    Rectangle (400,130 300x20), "Maximal start time [s]"
    Rectangle (400,150 300x20), "Set pressure to start [bar]"
    Rectangle (400,170 300x20), "Minimal presure increase [bar]"
    Rectangle (400,210 300x20), "Maxmial diffrence in presure [bar]"
    Rectangle (400,190 300x20), "Presure valve turn off [bar]"
    Rectangle (400,250 400x20), "Cycli x70 Test"
    Rectangle (0,250 400x20), "Cycli x30 Test"
    Rectangle (0,350 300x20), "Current limit [A]"
    Rectangle (0,270 300x20), "Cycle time [s]"
    Rectangle (0,290 300x20), "Cooling time [s]"
    Rectangle (0,310 300x20), "Presure to obtain [bar]"
    Rectangle (0,330 300x20), "Set presure to start [bar]"
    Checkbox (200,375 200x30), "Check start presure", variable: stChamberTestParams.bCheckStartPresureCycle30
    Rectangle (400,370 200x40)
    Rectangle (400,350 300x20), "Current limit [A]"
    Rectangle (400,270 300x20), "Cycle time [s]"
    Rectangle (400,290 300x20), "Cooling time [s]"
    Rectangle (400,310 300x20), "Presure to obtain [bar]"
    Rectangle (400,330 300x20), "Set presure to start [bar]"
    Checkbox (400,375 200x30), "Check start presure", variable: stChamberTestParams.bCheckStartPresureCycle70
    Rectangle (300,50 100x20), "%.1f", text variable: stChamberTestParams.rTest300SecTime
        OnMouseClick: write the text variable via Default, min 0, max 10000000
    Rectangle (300,70 100x20), "%.1f", text variable: stChamberTestParams.rPresureToObtainPerformanceTest
        OnMouseClick: write the text variable via Default, min 0, max 10
    Rectangle (300,90 100x20), "%.1f", text variable: stChamberTestParams.rCurrentLimitPerformacneTest
        OnMouseClick: write the text variable via Default, min 1, max 20
    Rectangle (300,190 100x20), "%.1f", text variable: stChamberTestParams.rTestHourTime
        OnMouseClick: write the text variable via Default, min 0, max 10000000
    Rectangle (300,210 100x20), "%.1f", text variable: stChamberTestParams.rPressureToObtainHourTest
        OnMouseClick: write the text variable via Default, min 0, max 10
    Rectangle (300,230 100x20), "%.1f", text variable: stChamberTestParams.rTestHourPressureMaximalTolerance
        OnMouseClick: write the text variable via Default, min 0, max 10
    Rectangle (700,50 100x20), "%.1f", text variable: stChamberTestParams.rTestCoolingTimeFullStepI
        OnMouseClick: write the text variable via Default, min 0, max 10000000
    Rectangle (700,70 100x20), "%.1f", text variable: stChamberTestParams.rTestCoolingTimeFullStepII
        OnMouseClick: write the text variable via Default, min 0, max 10000000
    Rectangle (700,150 100x20), "%.1f", text variable: stChamberTestParams.rTestUnderPresureSetPresure
        OnMouseClick: write the text variable via Default, min 0, max 10
    Rectangle (700,130 100x20), "%.1f", text variable: stChamberTestParams.rTestUnderPresureTime
        OnMouseClick: write the text variable via Default, min 0, max 10000000
    Rectangle (700,170 100x20), "%.1f", text variable: stChamberTestParams.rTestUnderPresureMinimalIncrease
        OnMouseClick: write the text variable via Default, min 0, max 10
    Rectangle (700,210 100x20), "%.1f", text variable: stChamberTestParams.rTestUnderPresureStartTolerance
        OnMouseClick: write the text variable via Default, min 0, max 10
    Rectangle (700,190 100x20), "%.1f", text variable: stChamberTestParams.rTestUnderPresureCloseTolerance
        OnMouseClick: write the text variable via Default, min 0, max 10
    Rectangle (300,350 100x20), "%.1f", text variable: stChamberTestParams.rCurrentLimitCycle30
        OnMouseClick: write the text variable via Default, min 0, max 10
    Rectangle (300,310 100x20), "%.1f", text variable: stChamberTestParams.rPresureToObtainCycle30Test
        OnMouseClick: write the text variable via Default, min 0, max 10
    Rectangle (300,330 100x20), "%.1f", text variable: stChamberTestParams.rStartPresureCycle30Test
        OnMouseClick: write the text variable via Default, min 0, max 10
    Rectangle (300,270 100x20), "%.1f", text variable: stChamberTestParams.rTestCycle30LimitTime
        OnMouseClick: write the text variable via Default, min 0, max 10000000
    Rectangle (300,290 100x20), "%.1f", text variable: stChamberTestParams.rTestCycle30CoolingTime
        OnMouseClick: write the text variable via Default, min 0, max 10000000
    Rectangle (700,350 100x20), "%.1f", text variable: stChamberTestParams.rCurrentLimitCycle70
        OnMouseClick: write the text variable via Default, min 0, max 10
    Rectangle (700,310 100x20), "%.1f", text variable: stChamberTestParams.rPresureToObtainCycle70Test
        OnMouseClick: write the text variable via Default, min 0, max 10
    Rectangle (700,330 100x20), "%.1f", text variable: stChamberTestParams.rStartPresureCycle70Test
        OnMouseClick: write the text variable via Default, min 0, max 10
    Rectangle (700,270 100x20), "%.1f", text variable: stChamberTestParams.rTestCycle70LimitTime
        OnMouseClick: write the text variable via Default, min 0, max 10000000
    Rectangle (700,290 100x20), "%.1f", text variable: stChamberTestParams.rTestCycle70CoolingTime
        OnMouseClick: write the text variable via Default, min 0, max 10000000
    Rectangle (300,130 100x20), "%.1f", text variable: stChamberTestParams.rTestEolLimitTime
        OnMouseClick: write the text variable via Default, min 0, max 10000000
    Rectangle (300,150 100x20), "%.1f", text variable: stChamberTestParams.rPresureToObtainEOLTest
        OnMouseClick: write the text variable via Default, min 0, max 10
    Rectangle (0,370 200x20), "Minimal current [A]"
    Rectangle (0,390 200x20), "%.1f", text variable: stChamberTestParams.rMinimalCurrentLimit
        OnMouseClick: write the text variable via Default, min 0, max 10
    Rectangle (600,370 200x20), "Minimal current check time [s]"
    Rectangle (600,390 200x20), "%.1f", text variable: stChamberTestParams.rMinimalCurrentCheckDelay
        OnMouseClick: write the text variable via Default, min 0, max 10
END_VISUALIZATION

// ---- QATester/VISUs/Screens/HMI/vMainScreen.TcVIS
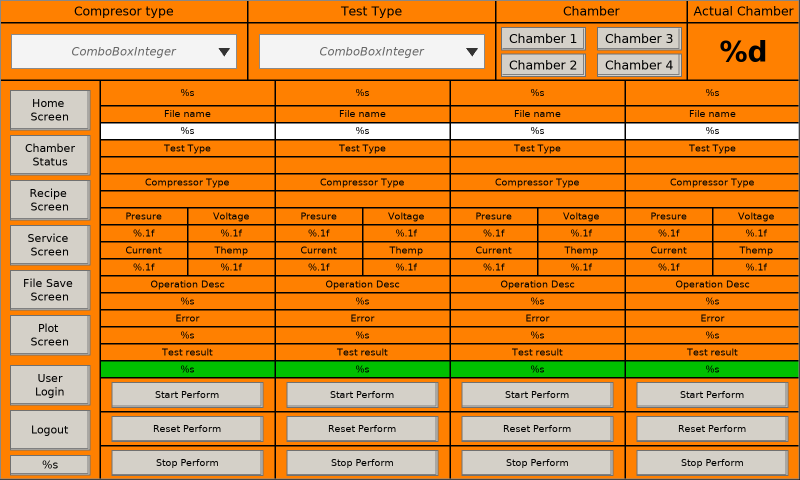
VISUALIZATION vMainScreen  // 800x480
VAR_IN_OUT
	arChamber : 	ARRAY[0..3] OF fbChamber;
	arParams :   ARRAY[0..3] OF stParamsChamber;
	arControl :   ARRAY[0..3] OF stControl;
	arTestParams : ARRAY[0..3] OF stTestParams;
END_VAR
VAR
	iActualChamber : INT;
	bLogin			: BOOL;
END_VAR
    Frame (0,0 800x80)
        shows vTestPicker(iCompressorPick := arParams[iActualChamber].iCompresorType, iTestType := arControl[iActualChamber].iSetTest, iActualChamber := iActualChamber, arControl := arControl)
    Frame (100,80 700x400)
        shows vStatusScreen(arChamber := arChamber, arParams := arParams, arControl := arControl)
        shows vRecipe(fbChamber := arChamber[iActualChamber], stChamberTestParams := arTestParams[arParams[iActualChamber].iCompresorType])
        shows vService(fbChamber := arChamber[iActualChamber], stParams := arParams[iActualChamber])
        shows vFileSave(fbChamber := arChamber[iActualChamber], stParams := arParams[iActualChamber])
        shows vPlotScreen(stControl := arControl[iActualChamber], fbChamber := arChamber[iActualChamber])
        shows vStatusScreen_v2(arChamber := arChamber[iActualChamber], arParams := arParams[iActualChamber], arControl := arControl[iActualChamber])
    Rectangle (0,80 100x400)
    Button (10,90 80x40), "Home Screen"
        OnMouseClick: FrameSelectionChange Selection=SelectedFrame=4e77f9b9-a257-46d1-860a-d32039bd6f78, GlobSel=IndExpr=4, AssignDir=vMainScreen.GenElemInst_5, AssignType=Directly, SelType=Locally
    Button (10,180 80x40), "Recipe Screen"
        OnMouseClick: FrameSelectionChange Selection=SelectedFrame=4e77f9b9-a257-46d1-860a-d32039bd6f78, Selection=1, GlobSel=IndExpr=1, AssignDir=vMainScreen.GenElemInst_5, AssignType=Directly, SelType=Locally
    Button (10,270 80x40), "File Save Screen"
        OnMouseClick: FrameSelectionChange Selection=SelectedFrame=4e77f9b9-a257-46d1-860a-d32039bd6f78, Selection=3, GlobSel=IndExpr=3, AssignDir=vMainScreen.GenElemInst_5, AssignType=Directly, SelType=Locally
    Button (10,225 80x40), "Service Screen"
        OnMouseClick: FrameSelectionChange Selection=SelectedFrame=4e77f9b9-a257-46d1-860a-d32039bd6f78, Selection=2, GlobSel=IndExpr=2, AssignDir=vMainScreen.GenElemInst_5, AssignType=Directly, SelType=Locally
    Button (10,315 80x40), "Plot Screen"
        OnMouseClick: FrameSelectionChange Selection=SelectedFrame=4e77f9b9-a257-46d1-860a-d32039bd6f78, Selection=4, GlobSel=IndExpr=4, AssignDir=vMainScreen.GenElemInst_5, AssignType=Directly, SelType=Locally
    Button (10,365 80x40), "User Login", pressed state: bLogin
        OnMouseClick: VisuUserMgmt Type=Login
    Button (10,410 80x40), "Logout", pressed state: bLogin
        OnMouseClick: VisuUserMgmt Type=Logout
    Button (10,455 80x20), "%s", text variable: Visu_Globals.CurrentUserGroupName, pressed state: bLogin
    Button (10,135 80x40), "Chamber Status"
        OnMouseClick: FrameSelectionChange Selection=SelectedFrame=4e77f9b9-a257-46d1-860a-d32039bd6f78, Selection=5, GlobSel=IndExpr=4, AssignDir=vMainScreen.GenElemInst_5, AssignType=Directly, SelType=Locally
END_VISUALIZATION

// ---- QATester/VISUs/Screens/HMI/vStatusScreen.TcVIS
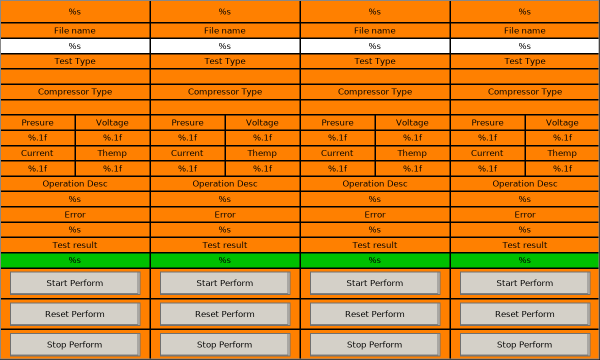
VISUALIZATION vStatusScreen  // 600x360
VAR_IN_OUT
	arChamber : 	ARRAY[0..3] OF fbChamber;
	arParams :   ARRAY[0..3] OF stParamsChamber;
	arControl :   ARRAY[0..3] OF stControl;
END_VAR
    Frame (0,0 150x360)
        shows vSmallChamber(stParams := arParams[0], fbChamber := arChamber[0], stControl := arControl[0])
    Frame (150,0 150x360)
        shows vSmallChamber(stParams := arParams[1], fbChamber := arChamber[1], stControl := arControl[1])
    Frame (450,0 150x360)
        shows vSmallChamber(stParams := arParams[3], fbChamber := arChamber[3], stControl := arControl[3])
    Frame (300,0 150x360)
        shows vSmallChamber(stParams := arParams[2], fbChamber := arChamber[2], stControl := arControl[2])
END_VISUALIZATION

// ---- QATester/VISUs/Screens/HMI/vStatusScreen_v2.TcVIS
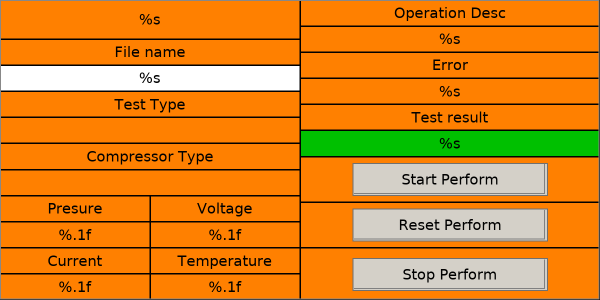
VISUALIZATION vStatusScreen_v2  // 600x300
VAR_IN_OUT
	arChamber :  fbChamber;
	arParams :    stParamsChamber;
	arControl :    stControl;
END_VAR
    Frame (0,0 600x300)
        shows vSmallChamber_v2(stParams := arParams, fbChamber := arChamber, stControl := arControl)
END_VISUALIZATION

// ---- QATester/VISUs/Screens/WEB/vMainScreen_WEB.TcVIS
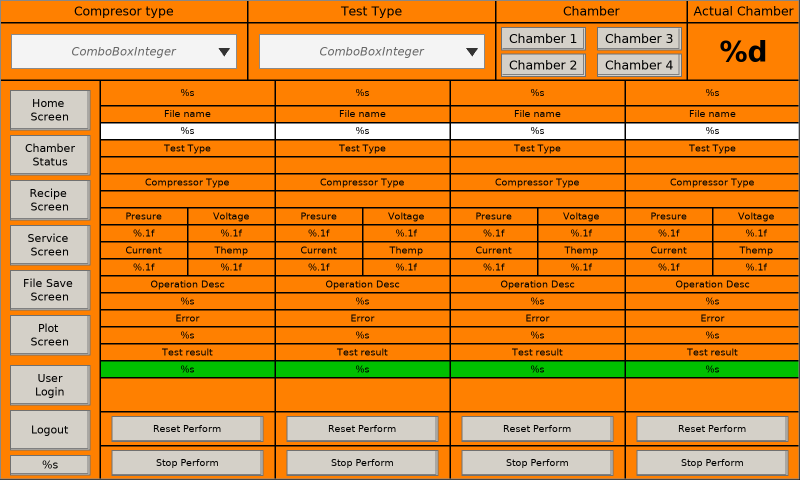
VISUALIZATION vMainScreen_WEB  // 800x480
VAR_IN_OUT
	arChamber : 	ARRAY[0..3] OF fbChamber;
	arParams :   ARRAY[0..3] OF stParamsChamber;
	arControl :   ARRAY[0..3] OF stControl;
	arTestParams : ARRAY[0..3] OF stTestParams;
END_VAR
VAR
	iActualChamber : INT;
	bLogin			: BOOL;
END_VAR
    Frame (0,0 800x80)
        shows vTestPicker(iCompressorPick := arParams[iActualChamber].iCompresorType, iTestType := arControl[iActualChamber].iSetTest, iActualChamber := iActualChamber, arControl := arControl)
    Frame (100,80 700x400)
        shows vStatusScreen_WEB(arChamber := arChamber, arParams := arParams, arControl := arControl)
        shows vRecipe(fbChamber := arChamber[iActualChamber], stChamberTestParams := arTestParams[arParams[iActualChamber].iCompresorType])
        shows vService(fbChamber := arChamber[iActualChamber], stParams := arParams[iActualChamber])
        shows vFileSave(fbChamber := arChamber[iActualChamber], stParams := arParams[iActualChamber])
        shows vPlotScreen(stControl := arControl[iActualChamber], fbChamber := arChamber[iActualChamber])
        shows vStatusScreen_v2_WEB(arChamber := arChamber[iActualChamber], arParams := arParams[iActualChamber], arControl := arControl[iActualChamber])
    Rectangle (0,80 100x400)
    Button (10,90 80x40), "Home Screen"
        OnMouseClick: FrameSelectionChange Selection=SelectedFrame=4e77f9b9-a257-46d1-860a-d32039bd6f78, GlobSel=IndExpr=4, AssignDir=vMainScreen.GenElemInst_5, AssignType=Directly, SelType=Locally
    Button (10,180 80x40), "Recipe Screen"
        OnMouseClick: FrameSelectionChange Selection=SelectedFrame=4e77f9b9-a257-46d1-860a-d32039bd6f78, Selection=1, GlobSel=IndExpr=1, AssignDir=vMainScreen.GenElemInst_5, AssignType=Directly, SelType=Locally
    Button (10,270 80x40), "File Save Screen"
        OnMouseClick: FrameSelectionChange Selection=SelectedFrame=4e77f9b9-a257-46d1-860a-d32039bd6f78, Selection=3, GlobSel=IndExpr=3, AssignDir=vMainScreen.GenElemInst_5, AssignType=Directly, SelType=Locally
    Button (10,225 80x40), "Service Screen"
        OnMouseClick: FrameSelectionChange Selection=SelectedFrame=4e77f9b9-a257-46d1-860a-d32039bd6f78, Selection=2, GlobSel=IndExpr=2, AssignDir=vMainScreen.GenElemInst_5, AssignType=Directly, SelType=Locally
    Button (10,315 80x40), "Plot Screen"
        OnMouseClick: FrameSelectionChange Selection=SelectedFrame=4e77f9b9-a257-46d1-860a-d32039bd6f78, Selection=4, GlobSel=IndExpr=4, AssignDir=vMainScreen.GenElemInst_5, AssignType=Directly, SelType=Locally
    Button (10,365 80x40), "User Login", pressed state: bLogin
        OnMouseClick: VisuUserMgmt Type=Login
    Button (10,410 80x40), "Logout", pressed state: bLogin
        OnMouseClick: VisuUserMgmt Type=Logout
    Button (10,455 80x20), "%s", text variable: Visu_Globals.CurrentUserGroupName, pressed state: bLogin
    Button (10,135 80x40), "Chamber Status"
        OnMouseClick: FrameSelectionChange Selection=SelectedFrame=4e77f9b9-a257-46d1-860a-d32039bd6f78, Selection=5, GlobSel=IndExpr=4, AssignDir=vMainScreen.GenElemInst_5, AssignType=Directly, SelType=Locally
END_VISUALIZATION

// ---- QATester/VISUs/Screens/WEB/vStatusScreen_v2_WEB.TcVIS
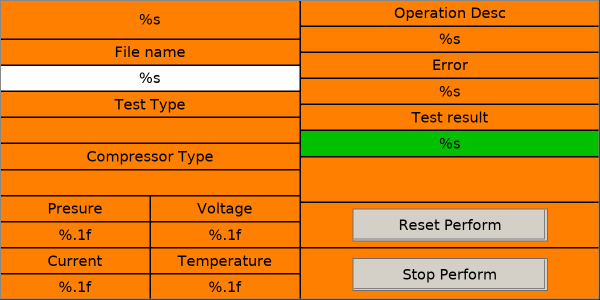
VISUALIZATION vStatusScreen_v2_WEB  // 600x300
VAR_IN_OUT
	arChamber :  fbChamber;
	arParams :    stParamsChamber;
	arControl :    stControl;
END_VAR
    Frame (0,0 600x300)
        shows vSmallChamber_v2_WEB(stParams := arParams, fbChamber := arChamber, stControl := arControl)
END_VISUALIZATION

// ---- QATester/VISUs/Screens/WEB/vStatusScreen_WEB.TcVIS
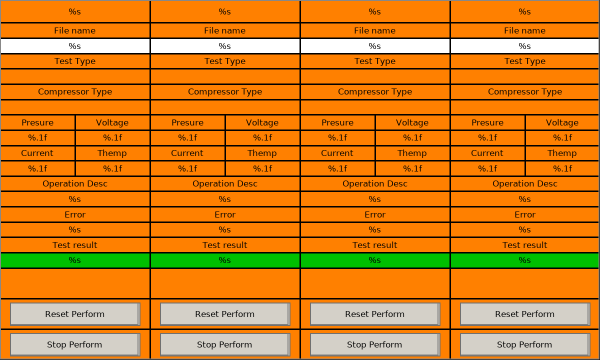
VISUALIZATION vStatusScreen_WEB  // 600x360
VAR_IN_OUT
	arChamber : 	ARRAY[0..3] OF fbChamber;
	arParams :   ARRAY[0..3] OF stParamsChamber;
	arControl :   ARRAY[0..3] OF stControl;
END_VAR
    Frame (0,0 150x360)
        shows vSmallChamber_WEB(stParams := arParams[0], fbChamber := arChamber[0], stControl := arControl[0])
    Frame (150,0 150x360)
        shows vSmallChamber_WEB(stParams := arParams[1], fbChamber := arChamber[1], stControl := arControl[1])
    Frame (450,0 150x360)
        shows vSmallChamber_WEB(stParams := arParams[3], fbChamber := arChamber[3], stControl := arControl[3])
    Frame (300,0 150x360)
        shows vSmallChamber_WEB(stParams := arParams[2], fbChamber := arChamber[2], stControl := arControl[2])
END_VISUALIZATION

// ---- QATester/VISUs/TextLists/txlCompresorTypes.TcTLO
TEXTLIST txlCompresorTypes
  1 = '8P0'
  2 = 'Volvo CMA'
   = ''
END_TEXTLIST

// ---- QATester/VISUs/TextLists/txlTestTypes.TcTLO
TEXTLIST txlTestTypes
  0 = 'none'
  10 = 'EOL'
  20 = 'Performance'
  30 = 'Hour'
  40 = 'Whole'
  50 = 'Cyclic 30'
  60 = 'Cyclic 70'
   = ''
END_TEXTLIST

// ---- QATester/VISUs/vMain.TcVIS
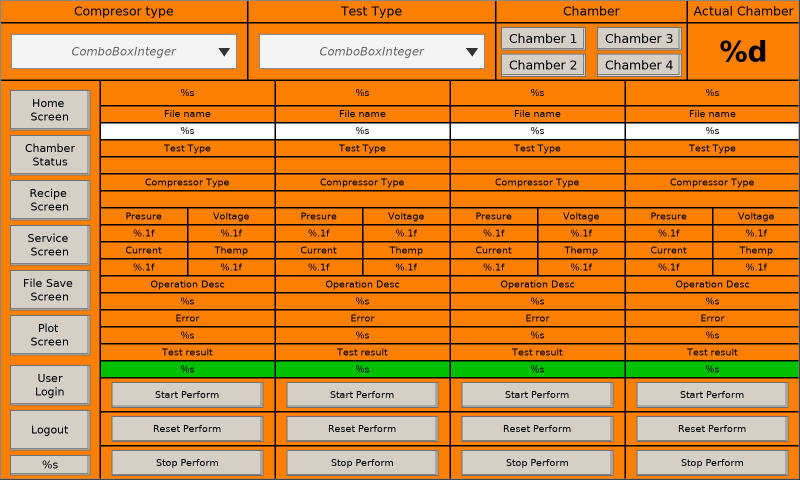
VISUALIZATION vMain  // 800x480
    Frame (0,0 800x480)
        shows vMainScreen(arChamber := MAIN.fb.arFbChamber, arParams := GVL_TesterParams.arstParams, arControl := GVL_TesterParams.arstControl, arTestParams := GVL_TesterParams.arTestParams)
        shows vRecipe(fbChamber := arChamber[iActualChamber], stChamberTestParams := arTestParams[arParams[iActualChamber].iCompresorType])
        shows vService(fbChamber := arChamber[iActualChamber], stParams := arParams[iActualChamber])
        shows vFileSave(fbChamber := arChamber[iActualChamber], stParams := arParams[iActualChamber])
        shows vPlotScreen(stControl := arControl[iActualChamber], fbChamber := arChamber[iActualChamber])
        shows vStatusScreen_v2(arChamber := arChamber[iActualChamber], arParams := arParams[iActualChamber], arControl := arControl[iActualChamber])
END_VISUALIZATION

// ---- QATester/VISUs/vMain_WEB.TcVIS
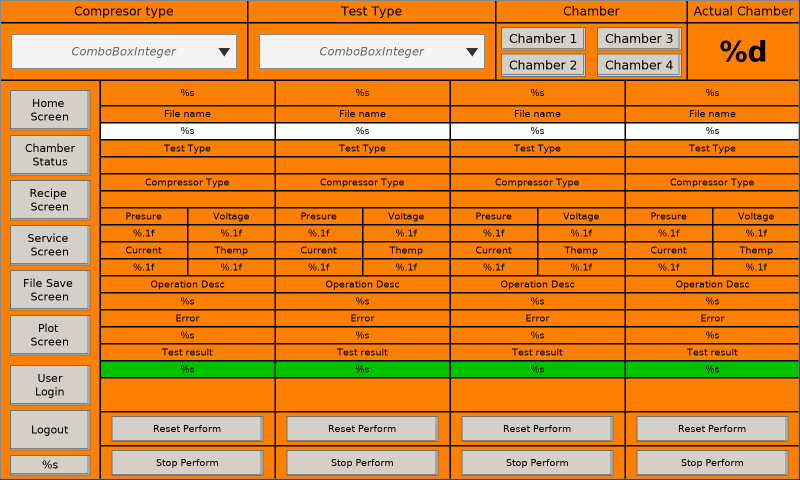
VISUALIZATION vMain_WEB  // 800x480
    Frame (0,0 800x480)
        shows vMainScreen_WEB(arChamber := MAIN.fb.arFbChamber, arParams := GVL_TesterParams.arstParams, arControl := GVL_TesterParams.arstControl, arTestParams := GVL_TesterParams.arTestParams)
        shows vService(fbChamber := arChamber[iActualChamber], stParams := arParams[iActualChamber])
        shows vFileSave(fbChamber := arChamber[iActualChamber], stParams := arParams[iActualChamber])
        shows vPlotScreen(stControl := arControl[iActualChamber], fbChamber := arChamber[iActualChamber])
        shows vStatusScreen_v2(arChamber := arChamber[iActualChamber], arParams := arParams[iActualChamber], arControl := arControl[iActualChamber])
        p2772295162: GVL_TesterParams.arTestParams
        p3795463443: GVL_TesterParams.arstControl
        p1849057978: GVL_TesterParams.arstParams
        p1287185654: MAIN.fb.arFbChamber
END_VISUALIZATION
